REGION Network 2: 0 - Запуск системы с нуля
   RUNG wire#powerrail
      Contact( #Start )
      { S7_Templates := "SrcType := Int" } EQ_Contact(in1 := #"Step", in2 := 0)
      wire#w1
      S_Coil( "PS_StartUp_DB".Start )
      wire#w2
      Contact( "PS_StartUp_DB".Ready )
      Add(in1 := #"Step", in2 := 1, out => #"Step")
      { S7_Templates := "SrcType := Int" } EQ_Contact(in1 := #Mode, in2 := 0)
      S_Coil( "PID_PE_DB".Start )
   END_RUNG
   RUNG wire#w2
      { S7_Templates := "SrcType := Int" } GT_Contact(in1 := "PS_StartUp_DB"."Step", in2 := 0)
      wire#w3
      { S7_Templates := "SrcType := Int" } EQ_Contact(in1 := #Mode, in2 := 1)
      S_Coil( "PID_LE_in_DB".Start )
   END_RUNG
   RUNG wire#w3
      { S7_Templates := "SrcType := Int" } EQ_Contact(in1 := #Mode, in2 := 2)
      S_Coil( "PID_LE_out_DB".Start )
   END_RUNG
   RUNG wire#w1
      { S7_Templates := "SrcType := Int" } EQ_Contact(in1 := #Mode, in2 := 0)
      Move(in := #PE_StartUp, out1 => #PE_Work)
      wire#w4
      { S7_Templates := "SrcType := Int" } GE_Contact(in1 := "PS_StartUp_DB"."Step", in2 := 1)
      R_Coil( "PID_PE_DB".CMD.Force )
   END_RUNG
   RUNG wire#w4
      { S7_Templates := "SrcType := Int" } LT_Contact(in1 := "PS_StartUp_DB"."Step", in2 := 1)
      Move(in := "PS_Main_DB".PS_SP_Hz, out1 => "PID_PE_DB".PID_Hand)
      S_Coil( "PID_PE_DB".CMD.Force )
   END_RUNG
   RUNG wire#w1
      { S7_Templates := "SrcType := Int" } LT_Contact(in1 := #PS_cnt, in2 := #PS_REQ)
      Move(in := "PS_Main_DB".PS_CMD, out1 => #PS_cnt, out2 => #PS_REQ)
   END_RUNG
   // the same network as SCL:
   #_w1 := #Start AND (#"Step" = 0);
   IF #_w1 THEN "PS_StartUp_DB".Start := TRUE; END_IF;
   #_w2 := #_w1 AND "PS_StartUp_DB".Ready;
   IF #_w2 THEN #"Step" := #"Step" + 1; END_IF;
   IF #_w2 AND (#Mode = 0) THEN "PID_PE_DB".Start := TRUE; END_IF;
   #_w3 := #_w1 AND ("PS_StartUp_DB"."Step" > 0);
   IF #_w3 AND (#Mode = 1) THEN "PID_LE_in_DB".Start := TRUE; END_IF;
   IF #_w3 AND (#Mode = 2) THEN "PID_LE_out_DB".Start := TRUE; END_IF;
   #_w4 := #_w1 AND (#Mode = 0);
   IF #_w4 THEN #PE_Work := #PE_StartUp; END_IF;
   IF #_w4 AND ("PS_StartUp_DB"."Step" >= 1) THEN "PID_PE_DB".CMD.Force := FALSE; END_IF;
   IF #_w4 AND ("PS_StartUp_DB"."Step" < 1) THEN
       "PID_PE_DB".PID_Hand := "PS_Main_DB".PS_SP_Hz;
       "PID_PE_DB".CMD.Force := TRUE;
   END_IF;
   IF #_w1 AND (#PS_cnt < #PS_REQ) THEN
       #PS_cnt := "PS_Main_DB".PS_CMD;
       #PS_REQ := "PS_Main_DB".PS_CMD;
   END_IF;
END_REGION

REGION Network 3: 1 - Штатная работа системы
   RUNG wire#powerrail
      { S7_Templates := "SrcType := Int" } EQ_Contact(in1 := #"Step", in2 := 1)
      { S7_Templates := "SrcType := Int" } LE_Contact(in1 := #Mode, in2 := 2)
      wire#w1
      { S7_Templates := "SrcType := Real" } GE_Contact(in1 := #SP_Hz, in2 := #SP_High)
      { S7_Templates := "SrcType := Int" } EQ_Contact(in1 := #PS_REQ, in2 := #PS_cnt)
      wire#w2
      { S7_Templates := "SrcType := Int" } LT_Contact(in1 := "PS_Main_DB".PS_CMD, in2 := "PS_Main_DB".PS_Group)
      { S7_Templates := "SrcType := Int" } LT_Contact(in1 := #PS_REQ, in2 := "PS_Main_DB".PS_Group)
      { S7_Templates := "SrcType := Int" } EQ_Contact(in1 := "PS_cnt_DB"."Step", in2 := 10)
      Coil( #T_Delay_ADD.Start )
      Contact( #T_Delay_ADD."Exit" )
      Add(in1 := #PS_REQ, in2 := 1, out => #PS_REQ)
   END_RUNG
   RUNG wire#w2
      I_Contact( #Reload )
      I_Contact( #Load )
      I_Contact( #Rotation )
      I_Contact( #Deload )
      I_Contact( #T_Delay_ADD."Exit" )
      { S7_Templates := "SrcType := Int" } EQ_Contact(in1 := "PS_cnt_DB"."Step", in2 := 10)
      Coil( #T_Delay_SUB.Start )
      Contact( #T_Delay_SUB."Exit" )
      wire#w3
      { S7_Templates := "SrcType := Int" } GT_Contact(in1 := #PS_REQ, in2 := "PS_Main_DB".PS_CMD)
      S_Coil( #Reload )
   END_RUNG
   RUNG wire#w3
      { S7_Templates := "SrcType := Int" } GT_Contact(in1 := "PS_Main_DB".PS_CMD, in2 := #PS_REQ)
      S_Coil( #Deload )
   END_RUNG
   RUNG wire#w1
      { S7_Templates := "SrcType := Real" } LT_Contact(in1 := #SP_Hz, in2 := #SP_Low)
      { S7_Templates := "SrcType := Int" } EQ_Contact(in1 := #PS_REQ, in2 := #PS_cnt)
      { S7_Templates := "SrcType := Int" } GT_Contact(in1 := #PS_REQ, in2 := 1)
      { S7_Templates := "SrcType := Int" } EQ_Contact(in1 := "PS_cnt_DB"."Step", in2 := 10)
      Sub(in1 := #PS_REQ, in2 := 1, out => #PS_REQ)
   END_RUNG
   RUNG wire#w1
      Move(in := #PE_SP, out1 => #PE_Work)
   END_RUNG
   // the same network as SCL:
   #_w1 := (#"Step" = 1) AND (#Mode <= 2);
   #_w2 := #_w1 AND (#SP_Hz >= #SP_High) AND (#PS_REQ = #PS_cnt);
   #T_Delay_ADD.Start := #_w2 AND ("PS_Main_DB".PS_CMD < "PS_Main_DB".PS_Group) AND (#PS_REQ < "PS_Main_DB".PS_Group) AND ("PS_cnt_DB"."Step" = 10);
   IF #T_Delay_ADD.Start AND #T_Delay_ADD."Exit" THEN #PS_REQ := #PS_REQ + 1; END_IF;
   #T_Delay_SUB.Start := #_w2 AND NOT #Reload AND NOT #Load AND NOT #Rotation AND NOT #Deload AND NOT #T_Delay_ADD."Exit" AND ("PS_cnt_DB"."Step" = 10);
   #_w3 := #T_Delay_SUB.Start AND #T_Delay_SUB."Exit";
   IF #_w3 AND (#PS_REQ > "PS_Main_DB".PS_CMD) THEN #Reload := TRUE; END_IF;
   IF #_w3 AND ("PS_Main_DB".PS_CMD > #PS_REQ) THEN #Deload := TRUE; END_IF;
   IF #_w1 AND (#SP_Hz < #SP_Low) AND (#PS_REQ = #PS_cnt) AND (#PS_REQ > 1) AND ("PS_cnt_DB"."Step" = 10) THEN
       #PS_REQ := #PS_REQ - 1;
   END_IF;
   IF #_w1 THEN #PE_Work := #PE_SP; END_IF;
END_REGION

REGION Network 4: 1 - Штатная работа - макс производительность
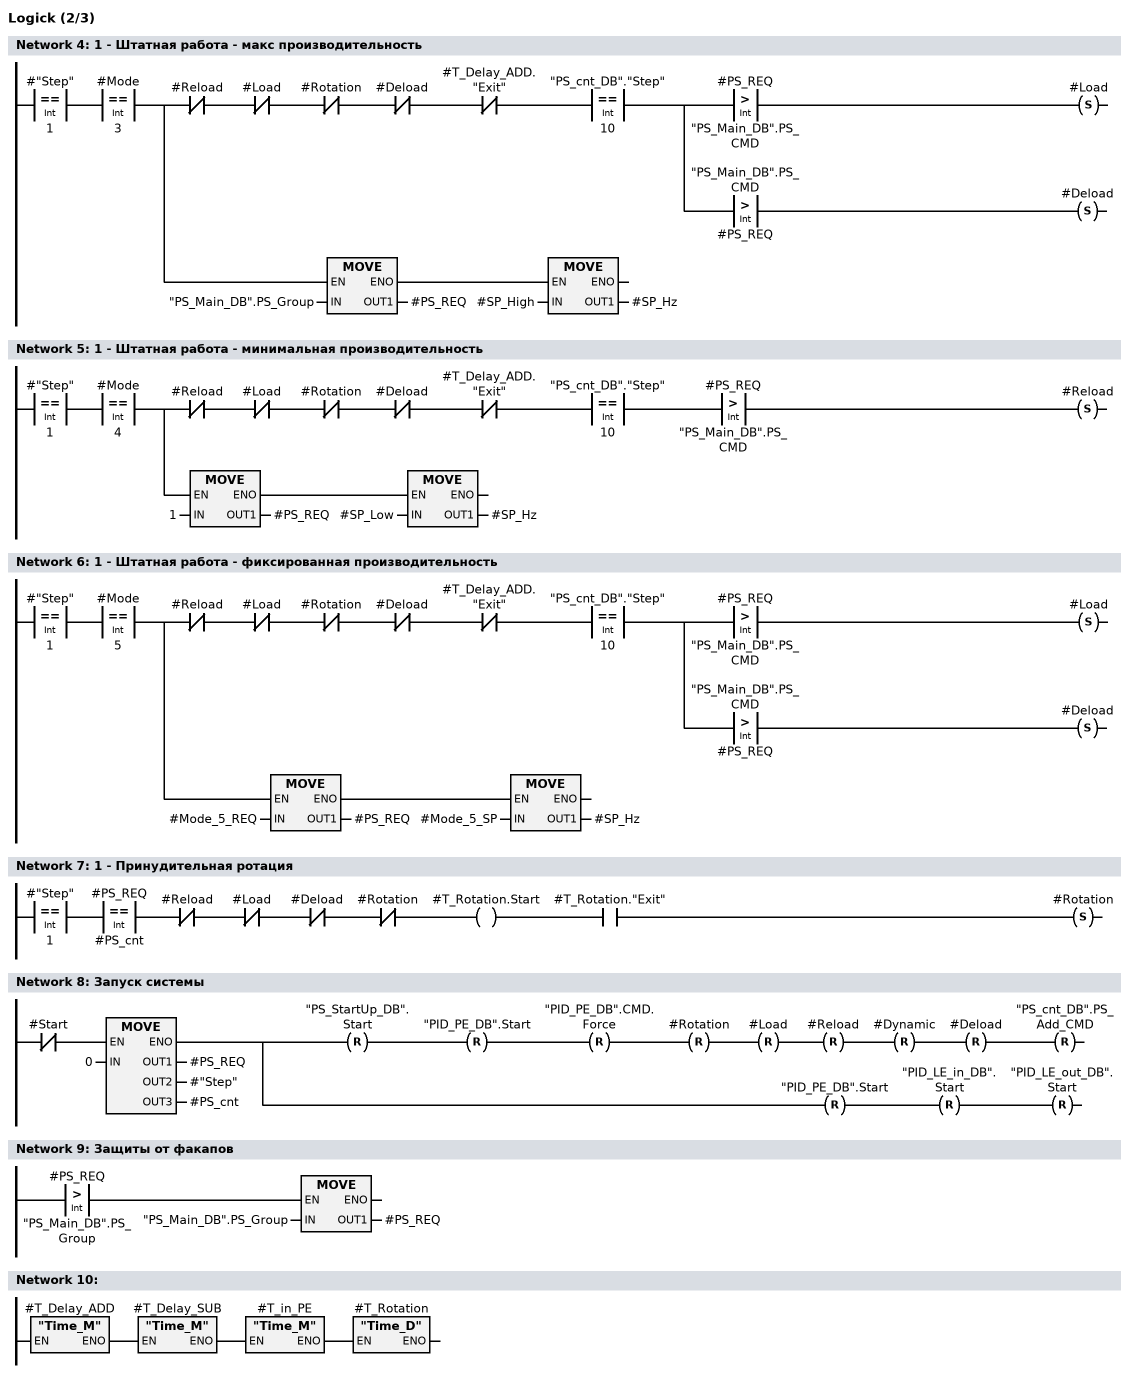
   RUNG wire#powerrail
      { S7_Templates := "SrcType := Int" } EQ_Contact(in1 := #"Step", in2 := 1)
      { S7_Templates := "SrcType := Int" } EQ_Contact(in1 := #Mode, in2 := 3)
      wire#w1
      I_Contact( #Reload )
      I_Contact( #Load )
      I_Contact( #Rotation )
      I_Contact( #Deload )
      I_Contact( #T_Delay_ADD."Exit" )
      { S7_Templates := "SrcType := Int" } EQ_Contact(in1 := "PS_cnt_DB"."Step", in2 := 10)
      wire#w2
      { S7_Templates := "SrcType := Int" } GT_Contact(in1 := #PS_REQ, in2 := "PS_Main_DB".PS_CMD)
      S_Coil( #Load )
   END_RUNG
   RUNG wire#w2
      { S7_Templates := "SrcType := Int" } GT_Contact(in1 := "PS_Main_DB".PS_CMD, in2 := #PS_REQ)
      S_Coil( #Deload )
   END_RUNG
   RUNG wire#w1
      Move(in := "PS_Main_DB".PS_Group, out1 => #PS_REQ)
      Move(in := #SP_High, out1 => #SP_Hz)
   END_RUNG
   // the same network as SCL:
   #_w1 := (#"Step" = 1) AND (#Mode = 3);
   #_w2 := #_w1 AND NOT #Reload AND NOT #Load AND NOT #Rotation AND NOT #Deload AND NOT #T_Delay_ADD."Exit" AND ("PS_cnt_DB"."Step" = 10);
   IF #_w2 AND (#PS_REQ > "PS_Main_DB".PS_CMD) THEN #Load := TRUE; END_IF;
   IF #_w2 AND ("PS_Main_DB".PS_CMD > #PS_REQ) THEN #Deload := TRUE; END_IF;
   IF #_w1 THEN
       #PS_REQ := "PS_Main_DB".PS_Group;
       #SP_Hz := #SP_High;
   END_IF;
END_REGION

REGION Network 5: 1 - Штатная работа - минимальная производительность
   RUNG wire#powerrail
      { S7_Templates := "SrcType := Int" } EQ_Contact(in1 := #"Step", in2 := 1)
      { S7_Templates := "SrcType := Int" } EQ_Contact(in1 := #Mode, in2 := 4)
      wire#w1
      I_Contact( #Reload )
      I_Contact( #Load )
      I_Contact( #Rotation )
      I_Contact( #Deload )
      I_Contact( #T_Delay_ADD."Exit" )
      { S7_Templates := "SrcType := Int" } EQ_Contact(in1 := "PS_cnt_DB"."Step", in2 := 10)
      { S7_Templates := "SrcType := Int" } GT_Contact(in1 := #PS_REQ, in2 := "PS_Main_DB".PS_CMD)
      S_Coil( #Reload )
   END_RUNG
   RUNG wire#w1
      Move(in := 1, out1 => #PS_REQ)
      Move(in := #SP_Low, out1 => #SP_Hz)
   END_RUNG
   // the same network as SCL:
   #_w1 := (#"Step" = 1) AND (#Mode = 4);
   IF #_w1 AND NOT #Reload AND NOT #Load AND NOT #Rotation AND NOT #Deload AND NOT #T_Delay_ADD."Exit" AND ("PS_cnt_DB"."Step" = 10) AND (#PS_REQ > "PS_Main_DB".PS_CMD) THEN
       #Reload := TRUE;
   END_IF;
   IF #_w1 THEN
       #PS_REQ := 1;
       #SP_Hz := #SP_Low;
   END_IF;
END_REGION

REGION Network 6: 1 - Штатная работа - фиксированная производительность
   RUNG wire#powerrail
      { S7_Templates := "SrcType := Int" } EQ_Contact(in1 := #"Step", in2 := 1)
      { S7_Templates := "SrcType := Int" } EQ_Contact(in1 := #Mode, in2 := 5)
      wire#w1
      I_Contact( #Reload )
      I_Contact( #Load )
      I_Contact( #Rotation )
      I_Contact( #Deload )
      I_Contact( #T_Delay_ADD."Exit" )
      { S7_Templates := "SrcType := Int" } EQ_Contact(in1 := "PS_cnt_DB"."Step", in2 := 10)
      wire#w2
      { S7_Templates := "SrcType := Int" } GT_Contact(in1 := #PS_REQ, in2 := "PS_Main_DB".PS_CMD)
      S_Coil( #Load )
   END_RUNG
   RUNG wire#w2
      { S7_Templates := "SrcType := Int" } GT_Contact(in1 := "PS_Main_DB".PS_CMD, in2 := #PS_REQ)
      S_Coil( #Deload )
   END_RUNG
   RUNG wire#w1
      Move(in := #Mode_5_REQ, out1 => #PS_REQ)
      Move(in := #Mode_5_SP, out1 => #SP_Hz)
   END_RUNG
   // the same network as SCL:
   #_w1 := (#"Step" = 1) AND (#Mode = 5);
   #_w2 := #_w1 AND NOT #Reload AND NOT #Load AND NOT #Rotation AND NOT #Deload AND NOT #T_Delay_ADD."Exit" AND ("PS_cnt_DB"."Step" = 10);
   IF #_w2 AND (#PS_REQ > "PS_Main_DB".PS_CMD) THEN #Load := TRUE; END_IF;
   IF #_w2 AND ("PS_Main_DB".PS_CMD > #PS_REQ) THEN #Deload := TRUE; END_IF;
   IF #_w1 THEN
       #PS_REQ := #Mode_5_REQ;
       #SP_Hz := #Mode_5_SP;
   END_IF;
END_REGION

REGION Network 7: 1 - Принудительная ротация
   RUNG wire#powerrail
      { S7_Templates := "SrcType := Int" } EQ_Contact(in1 := #"Step", in2 := 1)
      { S7_Templates := "SrcType := Int" } EQ_Contact(in1 := #PS_REQ, in2 := #PS_cnt)
      I_Contact( #Reload )
      I_Contact( #Load )
      I_Contact( #Deload )
      I_Contact( #Rotation )
      Coil( #T_Rotation.Start )
      Contact( #T_Rotation."Exit" )
      S_Coil( #Rotation )
   END_RUNG
   // the same network as SCL:
   #T_Rotation.Start := (#"Step" = 1) AND (#PS_REQ = #PS_cnt) AND NOT #Reload AND NOT #Load AND NOT #Deload AND NOT #Rotation;
   IF #T_Rotation.Start AND #T_Rotation."Exit" THEN #Rotation := TRUE; END_IF;
END_REGION

REGION Network 8: Запуск системы
   RUNG wire#powerrail
      I_Contact( #Start )
      Move(in := 0, out1 => #PS_REQ, out2 => #"Step", out3 => #PS_cnt)
      wire#w1
      R_Coil( "PS_StartUp_DB".Start )
      R_Coil( "PID_PE_DB".Start )
      R_Coil( "PID_PE_DB".CMD.Force )
      R_Coil( #Rotation )
      R_Coil( #Load )
      R_Coil( #Reload )
      R_Coil( #Dynamic )
      R_Coil( #Deload )
      R_Coil( "PS_cnt_DB".PS_Add_CMD )
   END_RUNG
   RUNG wire#w1
      R_Coil( "PID_PE_DB".Start )
      R_Coil( "PID_LE_in_DB".Start )
      R_Coil( "PID_LE_out_DB".Start )
   END_RUNG
   // the same network as SCL:
   IF NOT #Start THEN
       #PS_REQ := 0;
       #"Step" := 0;
       #PS_cnt := 0;
       "PS_StartUp_DB".Start := FALSE;
       "PID_PE_DB".Start := FALSE;
       "PID_PE_DB".CMD.Force := FALSE;
       #Rotation := FALSE;
       #Load := FALSE;
       #Reload := FALSE;
       #Dynamic := FALSE;
       #Deload := FALSE;
       "PS_cnt_DB".PS_Add_CMD := FALSE;
       "PID_PE_DB".Start := FALSE;
       "PID_LE_in_DB".Start := FALSE;
       "PID_LE_out_DB".Start := FALSE;
   END_IF;
END_REGION

REGION Network 9: Защиты от факапов
   RUNG wire#powerrail
      { S7_Templates := "SrcType := Int" } GT_Contact(in1 := #PS_REQ, in2 := "PS_Main_DB".PS_Group)
      Move(in := "PS_Main_DB".PS_Group, out1 => #PS_REQ)
   END_RUNG
   // the same network as SCL:
   IF #PS_REQ > "PS_Main_DB".PS_Group THEN #PS_REQ := "PS_Main_DB".PS_Group; END_IF;
END_REGION

REGION Network 10
   RUNG wire#powerrail
      #T_Delay_ADD()
      #T_Delay_SUB()
      #T_in_PE()
      #T_Rotation()
   END_RUNG
   // the same network as SCL:
   #T_Delay_ADD(ENO => #_w1);   // "Time_M"
   #T_Delay_SUB(EN := #_w1, ENO => #_w2);   // "Time_M"
   #T_in_PE(EN := #_w2, ENO => #_w3);   // "Time_M"
   IF #_w3 THEN
       #T_Rotation();   // "Time_D"
   END_IF;
END_REGION

REGION Network 11: Соотношение давления к уставке
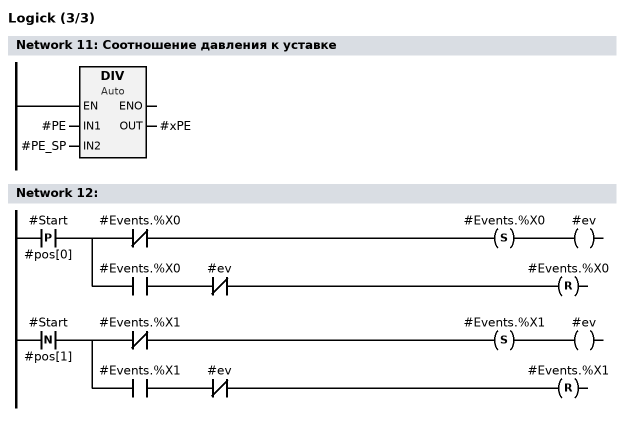
   RUNG wire#powerrail
      Div(in1 := #PE, in2 := #PE_SP, out => #xPE)
   END_RUNG
   // the same network as SCL:
   #xPE := #PE / #PE_SP;
END_REGION

REGION Network 12
   RUNG wire#powerrail
      P_Contact(operand := #Start, bit := #pos[0])
      wire#w1
      I_Contact( #Events.%X0 )
      S_Coil( #Events.%X0 )
      Coil( #ev )
   END_RUNG
   RUNG wire#w1
      Contact( #Events.%X0 )
      I_Contact( #ev )
      R_Coil( #Events.%X0 )
   END_RUNG
   RUNG wire#powerrail
      N_Contact(operand := #Start, bit := #pos[1])
      wire#w2
      I_Contact( #Events.%X1 )
      S_Coil( #Events.%X1 )
      Coil( #ev )
   END_RUNG
   RUNG wire#w2
      Contact( #Events.%X1 )
      I_Contact( #ev )
      R_Coil( #Events.%X1 )
   END_RUNG
   // the same network as SCL:
   #_w1 := #Start AND NOT #pos[0];   // rising edge of #Start
   #pos[0] := #Start;
   #_w2 := #_w1 AND NOT #Events.%X0;
   IF #_w2 THEN #Events.%X0 := TRUE; END_IF;
   #ev := #_w2;
   IF #_w1 AND #Events.%X0 AND NOT #ev THEN #Events.%X0 := FALSE; END_IF;
   #_w3 := NOT #Start AND #pos[1];   // falling edge of #Start
   #pos[1] := #Start;
   #_w4 := #_w3 AND NOT #Events.%X1;
   IF #_w4 THEN #Events.%X1 := TRUE; END_IF;
   #ev := #_w4;
   IF #_w3 AND #Events.%X1 AND NOT #ev THEN #Events.%X1 := FALSE; END_IF;
END_REGION
END_FUNCTION_BLOCK

FUNCTION_BLOCK "PS_Main"   // FB10, LAD
{ S7_Optimized_Access := 'FALSE' }
VERSION : 0.1
// stored: AutoNumber false, IsIECCheckEnabled false, SetENOAutomatically false, UDAEnableTagReadback false
   VAR_IN_OUT
      PS_REQ : Int;   // Требуемуе кол-во насосов
      PS_cnt : Int;
   END_VAR
   VAR DB_SPECIFIC
      Step_Up { S7_SetPoint := 'True'} : Array[1..6] of Real;   // Ускорения насоса, Гц/сек
      Step_Down { S7_SetPoint := 'True'} : Array[1..6] of Real;   // Замедление насоса, Гц/сек
   END_VAR
   VAR
      PS_One { S7_SetPoint := 'True'} : Array[0..10] of "PS_One";   // Pump System - One Pump
   END_VAR
   VAR DB_SPECIFIC
      PS_All { S7_SetPoint := 'True'} : Int := 7;   // Общее количество насосов
      PS_Group { S7_SetPoint := 'True'} : Int := 5;   // Число основных насосов
      PS_Reserv { S7_SetPoint := 'True'} : Int := 2;   // Число резервных насосов
      PS_Ready : Int;   // Число готовых насосов
      PS_CMD : Int;   // Число насосов в работе
      PS_Work : Int;   // Число штатно работающих насосов
      PS_Load : Int;   // Число нагруженных насосов
      PS_SP_Hz : Real;   // Уставка - штатная работа
      PS_Point : Real;
      PS_min_cnt : Int;   // Число замедленных насосов
   END_VAR
   VAR_TEMP   // added for the SCL form of the ladder/FBD networks
      _w1 : Bool;
   END_VAR
BEGIN

REGION Network 1: Распределение нагрузки по насосам
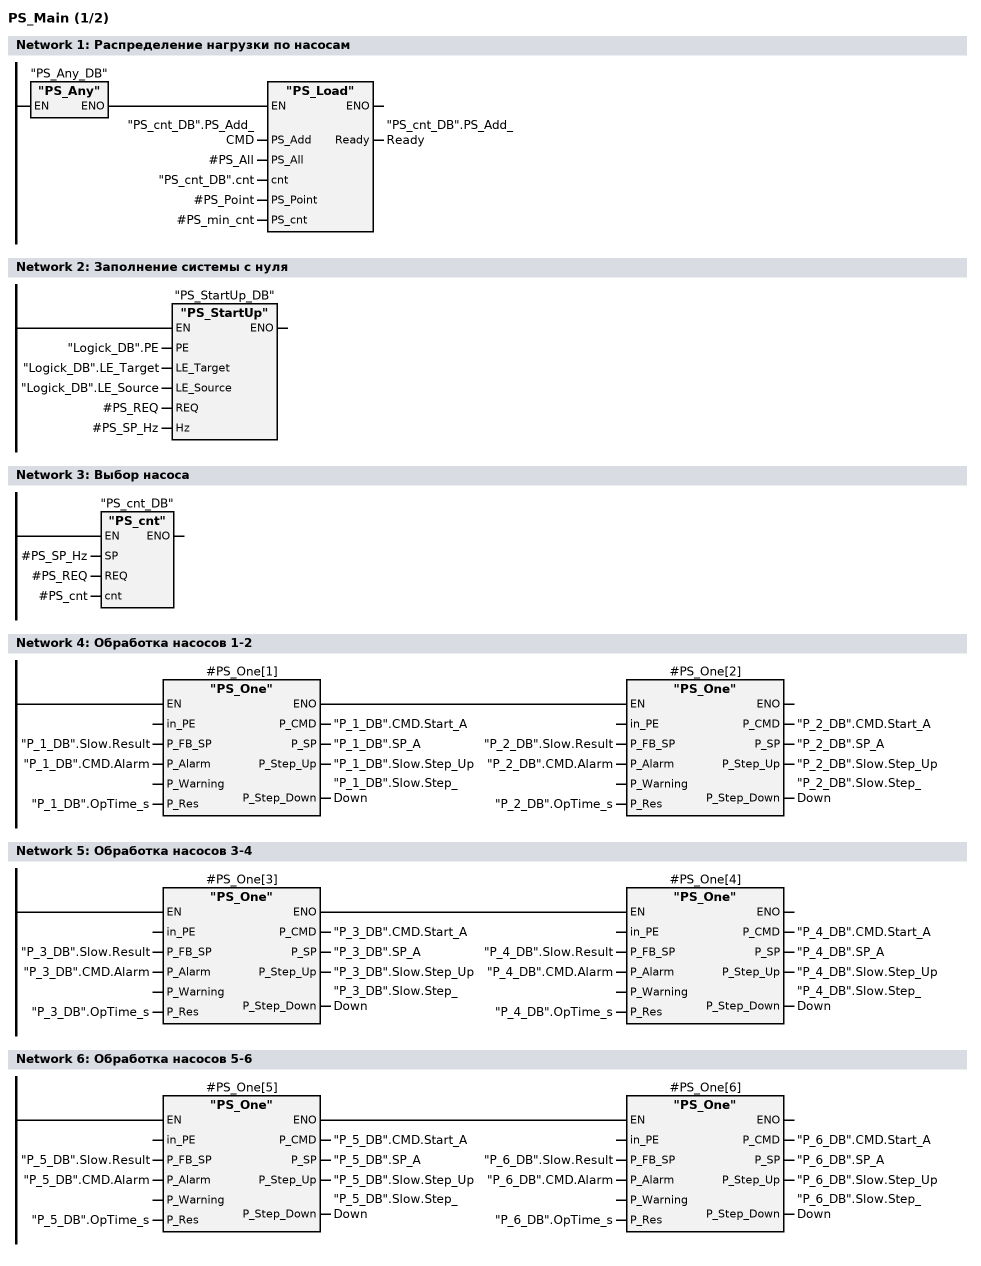
   RUNG wire#powerrail
      "PS_Any_DB"()
      "PS_Load"(PS_Add := "PS_cnt_DB".PS_Add_CMD, PS_All := #PS_All, cnt := "PS_cnt_DB".cnt, PS_Point := #PS_Point, PS_cnt := #PS_min_cnt, Ready => "PS_cnt_DB".PS_Add_Ready)
   END_RUNG
   // the same network as SCL:
   "PS_Any_DB"(ENO => #_w1);   // "PS_Any"
   IF #_w1 THEN
       "PS_Load"(PS_Add := "PS_cnt_DB".PS_Add_CMD,
                 PS_All := #PS_All,
                 cnt := "PS_cnt_DB".cnt,
                 PS_Point := #PS_Point,
                 PS_cnt := #PS_min_cnt,
                 Ready => "PS_cnt_DB".PS_Add_Ready);
   END_IF;
END_REGION

REGION Network 2: Заполнение системы с нуля
   RUNG wire#powerrail
      "PS_StartUp_DB"(PE := "Logick_DB".PE, LE_Target := "Logick_DB".LE_Target, LE_Source := "Logick_DB".LE_Source, REQ := #PS_REQ, Hz := #PS_SP_Hz)
   END_RUNG
   // the same network as SCL:
   "PS_StartUp_DB"(PE := "Logick_DB".PE,   // "PS_StartUp"
                   LE_Target := "Logick_DB".LE_Target,
                   LE_Source := "Logick_DB".LE_Source,
                   REQ := #PS_REQ,
                   Hz := #PS_SP_Hz);
END_REGION

REGION Network 3: Выбор насоса
   RUNG wire#powerrail
      "PS_cnt_DB"(SP := #PS_SP_Hz, REQ := #PS_REQ, cnt := #PS_cnt)
   END_RUNG
   // the same network as SCL:
   "PS_cnt_DB"(SP := #PS_SP_Hz, REQ := #PS_REQ, cnt := #PS_cnt);   // "PS_cnt"
END_REGION

REGION Network 4: Обработка насосов 1-2
   RUNG wire#powerrail
      #PS_One[1](in_PE :=, P_FB_SP := "P_1_DB".Slow.Result, P_Alarm := "P_1_DB".CMD.Alarm, P_Warning :=, P_Res := "P_1_DB".OpTime_s, P_CMD => "P_1_DB".CMD.Start_A, P_SP => "P_1_DB".SP_A, P_Step_Up => "P_1_DB".Slow.Step_Up, P_Step_Down => "P_1_DB".Slow.Step_Down)
      #PS_One[2](in_PE :=, P_FB_SP := "P_2_DB".Slow.Result, P_Alarm := "P_2_DB".CMD.Alarm, P_Warning :=, P_Res := "P_2_DB".OpTime_s, P_CMD => "P_2_DB".CMD.Start_A, P_SP => "P_2_DB".SP_A, P_Step_Up => "P_2_DB".Slow.Step_Up, P_Step_Down => "P_2_DB".Slow.Step_Down)
   END_RUNG
   // the same network as SCL:
   #PS_One[1](P_FB_SP := "P_1_DB".Slow.Result,   // "PS_One"
              P_Alarm := "P_1_DB".CMD.Alarm,
              P_Res := "P_1_DB".OpTime_s,
              P_CMD => "P_1_DB".CMD.Start_A,
              P_SP => "P_1_DB".SP_A,
              P_Step_Up => "P_1_DB".Slow.Step_Up,
              P_Step_Down => "P_1_DB".Slow.Step_Down,
              ENO => #_w1);
   IF #_w1 THEN
       #PS_One[2](P_FB_SP := "P_2_DB".Slow.Result,   // "PS_One"
                  P_Alarm := "P_2_DB".CMD.Alarm,
                  P_Res := "P_2_DB".OpTime_s,
                  P_CMD => "P_2_DB".CMD.Start_A,
                  P_SP => "P_2_DB".SP_A,
                  P_Step_Up => "P_2_DB".Slow.Step_Up,
                  P_Step_Down => "P_2_DB".Slow.Step_Down);
   END_IF;
END_REGION

REGION Network 5: Обработка насосов 3-4
   RUNG wire#powerrail
      #PS_One[3](in_PE :=, P_FB_SP := "P_3_DB".Slow.Result, P_Alarm := "P_3_DB".CMD.Alarm, P_Warning :=, P_Res := "P_3_DB".OpTime_s, P_CMD => "P_3_DB".CMD.Start_A, P_SP => "P_3_DB".SP_A, P_Step_Up => "P_3_DB".Slow.Step_Up, P_Step_Down => "P_3_DB".Slow.Step_Down)
      #PS_One[4](in_PE :=, P_FB_SP := "P_4_DB".Slow.Result, P_Alarm := "P_4_DB".CMD.Alarm, P_Warning :=, P_Res := "P_4_DB".OpTime_s, P_CMD => "P_4_DB".CMD.Start_A, P_SP => "P_4_DB".SP_A, P_Step_Up => "P_4_DB".Slow.Step_Up, P_Step_Down => "P_4_DB".Slow.Step_Down)
   END_RUNG
   // the same network as SCL:
   #PS_One[3](P_FB_SP := "P_3_DB".Slow.Result,   // "PS_One"
              P_Alarm := "P_3_DB".CMD.Alarm,
              P_Res := "P_3_DB".OpTime_s,
              P_CMD => "P_3_DB".CMD.Start_A,
              P_SP => "P_3_DB".SP_A,
              P_Step_Up => "P_3_DB".Slow.Step_Up,
              P_Step_Down => "P_3_DB".Slow.Step_Down,
              ENO => #_w1);
   IF #_w1 THEN
       #PS_One[4](P_FB_SP := "P_4_DB".Slow.Result,   // "PS_One"
                  P_Alarm := "P_4_DB".CMD.Alarm,
                  P_Res := "P_4_DB".OpTime_s,
                  P_CMD => "P_4_DB".CMD.Start_A,
                  P_SP => "P_4_DB".SP_A,
                  P_Step_Up => "P_4_DB".Slow.Step_Up,
                  P_Step_Down => "P_4_DB".Slow.Step_Down);
   END_IF;
END_REGION

REGION Network 6: Обработка насосов 5-6
   RUNG wire#powerrail
      #PS_One[5](in_PE :=, P_FB_SP := "P_5_DB".Slow.Result, P_Alarm := "P_5_DB".CMD.Alarm, P_Warning :=, P_Res := "P_5_DB".OpTime_s, P_CMD => "P_5_DB".CMD.Start_A, P_SP => "P_5_DB".SP_A, P_Step_Up => "P_5_DB".Slow.Step_Up, P_Step_Down => "P_5_DB".Slow.Step_Down)
      #PS_One[6](in_PE :=, P_FB_SP := "P_6_DB".Slow.Result, P_Alarm := "P_6_DB".CMD.Alarm, P_Warning :=, P_Res := "P_6_DB".OpTime_s, P_CMD => "P_6_DB".CMD.Start_A, P_SP => "P_6_DB".SP_A, P_Step_Up => "P_6_DB".Slow.Step_Up, P_Step_Down => "P_6_DB".Slow.Step_Down)
   END_RUNG
   // the same network as SCL:
   #PS_One[5](P_FB_SP := "P_5_DB".Slow.Result,   // "PS_One"
              P_Alarm := "P_5_DB".CMD.Alarm,
              P_Res := "P_5_DB".OpTime_s,
              P_CMD => "P_5_DB".CMD.Start_A,
              P_SP => "P_5_DB".SP_A,
              P_Step_Up => "P_5_DB".Slow.Step_Up,
              P_Step_Down => "P_5_DB".Slow.Step_Down,
              ENO => #_w1);
   IF #_w1 THEN
       #PS_One[6](P_FB_SP := "P_6_DB".Slow.Result,   // "PS_One"
                  P_Alarm := "P_6_DB".CMD.Alarm,
                  P_Res := "P_6_DB".OpTime_s,
                  P_CMD => "P_6_DB".CMD.Start_A,
                  P_SP => "P_6_DB".SP_A,
                  P_Step_Up => "P_6_DB".Slow.Step_Up,
                  P_Step_Down => "P_6_DB".Slow.Step_Down);
   END_IF;
END_REGION

REGION Network 7: Обработка насосов 7-8
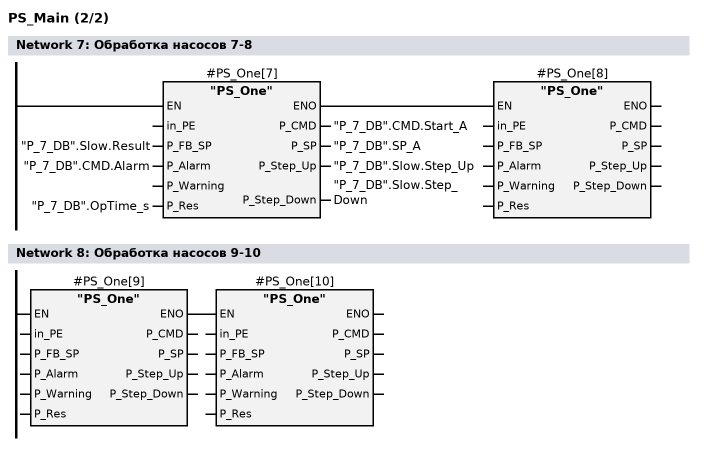
   RUNG wire#powerrail
      #PS_One[7](in_PE :=, P_FB_SP := "P_7_DB".Slow.Result, P_Alarm := "P_7_DB".CMD.Alarm, P_Warning :=, P_Res := "P_7_DB".OpTime_s, P_CMD => "P_7_DB".CMD.Start_A, P_SP => "P_7_DB".SP_A, P_Step_Up => "P_7_DB".Slow.Step_Up, P_Step_Down => "P_7_DB".Slow.Step_Down)
      #PS_One[8](in_PE :=, P_FB_SP :=, P_Alarm :=, P_Warning :=, P_Res :=, P_CMD =>, P_SP =>, P_Step_Up =>, P_Step_Down =>)
   END_RUNG
   // the same network as SCL:
   #PS_One[7](P_FB_SP := "P_7_DB".Slow.Result,   // "PS_One"
              P_Alarm := "P_7_DB".CMD.Alarm,
              P_Res := "P_7_DB".OpTime_s,
              P_CMD => "P_7_DB".CMD.Start_A,
              P_SP => "P_7_DB".SP_A,
              P_Step_Up => "P_7_DB".Slow.Step_Up,
              P_Step_Down => "P_7_DB".Slow.Step_Down,
              ENO => #_w1);
   IF #_w1 THEN
       #PS_One[8]();   // "PS_One"
   END_IF;
END_REGION

REGION Network 8: Обработка насосов 9-10
   RUNG wire#powerrail
      #PS_One[9](P_FB_SP :=, P_Alarm :=, P_Warning :=, P_Res :=, P_CMD =>, P_SP =>, P_Step_Up =>, P_Step_Down =>, in_PE :=)
      #PS_One[10](P_FB_SP :=, P_Alarm :=, P_Warning :=, P_Res :=, P_CMD =>, P_SP =>, P_Step_Up =>, P_Step_Down =>, in_PE :=)
   END_RUNG
   // the same network as SCL:
   #PS_One[9](ENO => #_w1);   // "PS_One"
   IF #_w1 THEN
       #PS_One[10]();   // "PS_One"
   END_IF;
END_REGION
END_FUNCTION_BLOCK

FUNCTION_BLOCK "PS_Any"
{ S7_Optimized_Access := 'FALSE' }
VERSION : 0.1
   VAR 
      x : Array[0..10] of Real;
      Delta_PE : Real;
      Delta_LE_in : Real;
      Delta_LE_out : Real;
   END_VAR


BEGIN
	//чтение уставки с ПИД-регулятора, если он в работе - режим работы по давлению
	IF "PID_PE_DB".Start AND NOT "PID_PE_DB".CMD.Hand AND "Logick_DB".Mode = 0 THEN
	    "Logick_DB".SP_Hz := "PID_PE_DB".Result;
	END_IF;
	
	//чтение уставки с ПИД-регулятора, если он в работе - режим работы по уровню в РЧВ
	IF "PID_LE_in_DB".Start AND NOT "PID_LE_in_DB".CMD.Hand AND "Logick_DB".Mode = 1 THEN
	    "Logick_DB".SP_Hz := "PID_LE_in_DB".Result;
	    IF "PS_StartUp_DB".Step = 1 THEN
	        "Logick_DB".SP_Hz := "Logick_DB".SP_Hz * "PS_StartUp_DB".xTime[2].Progress;
	    END_IF;
	END_IF;
	
	//чтение уставки с ПИД-регулятора, если он в работе - режим работы по уровню в городе
	IF "PID_LE_out_DB".Start AND NOT "PID_LE_out_DB".CMD.Hand AND "Logick_DB".Mode = 2 THEN
	    "Logick_DB".SP_Hz := "PID_LE_out_DB".Result;
	    IF "PS_StartUp_DB".Step = 1 THEN
	        "Logick_DB".SP_Hz := "Logick_DB".SP_Hz * "PS_StartUp_DB".xTime[2].Progress;
	    END_IF;
	END_IF;
	
	//рассчёт коррекции при превышении рабочего давления
	#x[1] := "Logick_DB".SP_PE_Alarm - "Logick_DB".SP_PE_Warning;
	#x[2] := "Logick_DB".PE - "Logick_DB".SP_PE_Warning;
	#x[3] := #x[2] / #x[1];
	#Delta_PE := 1 - #x[3];
	
	//давление выше рабочей точки
	IF #Delta_PE <= 1.0 THEN
	    "Logick_DB".PE_Warning := TRUE;
	    "Logick_DB".Alarms.%X0 := TRUE;
	ELSE
	    "Logick_DB".PE_Warning := FALSE;
	    "Logick_DB".Alarms.%X0 := FALSE;
	    #Delta_PE := 1.0;
	END_IF;
	
	//давление в аварийной зоне
	IF #Delta_PE <= 0.0 THEN
	    "Logick_DB".PE_Alarm := TRUE;
	    "Logick_DB".Alarms.%X1 := TRUE;
	    #Delta_PE := 0.0;
	ELSE
	    "Logick_DB".PE_Alarm := FALSE;
	END_IF;
	
	//рассчёт коррекции при падении уровня в РЧВ
	#x[4] := "Logick_DB".SP_LE_in_Warning - "Logick_DB".SP_LE_in_Alarm;
	#x[5] := "Logick_DB".LE_Source - "Logick_DB".SP_LE_in_Alarm;
	#x[6] := #x[5] / #x[4];
	#Delta_LE_in := #x[6];
	
	//уровень ниже рабочей точки
	IF #Delta_LE_in < 1.0 THEN
	    "Logick_DB".LE_in_Warning := TRUE;
	    "Logick_DB".Alarms.%X2 := TRUE;
	ELSE
	    "Logick_DB".LE_in_Warning := FALSE;
	    "Logick_DB".Alarms.%X2 := FALSE;
	    #Delta_LE_in := 1.0;
	END_IF;
	
	//уровень в аварийной зоне
	IF #Delta_LE_in <= 0.0 THEN
	    "Logick_DB".LE_in_Alarm := TRUE;
	    "Logick_DB".Alarms.%X3 := TRUE;
	    #Delta_LE_in := 0.0;
	ELSE
	    "Logick_DB".LE_in_Alarm := FALSE;
	END_IF;
	
	//рассчёт коррекции при превышении уровня в городе
	#x[7] := "Logick_DB".SP_LE_out_Alarm - "Logick_DB".SP_LE_out_Warning;
	#x[8] := "Logick_DB".LE_Target - "Logick_DB".SP_LE_out_Warning;
	#x[9] := #x[8] / #x[7];
	#Delta_LE_out := 1 - #x[9];
	
	//давление выше рабочей точки
	IF #Delta_LE_out <= 1.0 THEN
	    "Logick_DB".LE_out_Warning := TRUE;
	    "Logick_DB".Alarms.%X4 := TRUE;
	ELSE
	    "Logick_DB".LE_out_Warning := FALSE;
	    "Logick_DB".Alarms.%X4 := FALSE;
	    #Delta_LE_out := 1.0;
	END_IF;
	
	//давление в аварийной зоне
	IF #Delta_LE_out <= 0.0 THEN
	    "Logick_DB".LE_out_Alarm := TRUE;
	    "Logick_DB".Alarms.%X5 := TRUE;
	    #Delta_LE_out := 0.0;
	ELSE
	    "Logick_DB".LE_out_Alarm := FALSE;
	END_IF;
	
	//коррекция уставки при аварийных ситуациях
	"PS_Main_DB".PS_SP_Hz := "Logick_DB".SP_Hz * #Delta_PE * #Delta_LE_in * #Delta_LE_out;
	
	//Сброс аварий
	IF "Reset_All" THEN
	    "Logick_DB".Alarms := 0;
	END_IF;
	
	//индикатор аварий
	IF "Logick_DB".Alarms > 0 THEN
	    "Alm_Logick" := TRUE;
	END_IF;
	
END_FUNCTION_BLOCK

FUNCTION "PS_Load" : Void
{ S7_Optimized_Access := 'TRUE' }
VERSION : 0.1
   VAR_INPUT 
      PS_Add : Bool;
   END_VAR

   VAR_OUTPUT 
      Ready : Bool;
   END_VAR

   VAR_IN_OUT 
      PS_All : Int;
      cnt : Int;
      PS_Point : Real;   // точка схождения
      PS_cnt : Int;   // число готовых насосов
   END_VAR

   VAR_TEMP 
      x : Int;
   END_VAR


BEGIN
	//обнуление временных значений
	#PS_cnt := 0;
	#Ready := FALSE;
	"PS_cnt_DB".SP_High := "Logick_DB".SP_High;
	"PID_PE_DB".Settings.Max_out := "Logick_DB".SP_High + 1;
	"PID_PE_DB".Settings.Min_out := "Logick_DB".SP_Low - 1;
	"PID_LE_in_DB".Settings.Max_out := "Logick_DB".SP_High + 1;
	"PID_LE_in_DB".Settings.Min_out := "Logick_DB".SP_Low - 1;
	"PID_LE_out_DB".Settings.Max_out := "Logick_DB".SP_High + 1;
	"PID_LE_out_DB".Settings.Min_out := "Logick_DB".SP_Low - 1;
	"PS_cnt_DB".SP_Min := "Logick_DB".SP_Min;
	"Logick_DB".SP_Low := "PS_cnt_DB".SP_Low;
	"PS_Main_DB".PS_Ready := 0;
	"PS_Main_DB".PS_CMD := 0;
	"PS_Main_DB".PS_Work := 0;
	"PS_Main_DB".PS_Load := 0;
	
	IF "Logick_DB".SP_Hz > "Logick_DB".SP_High THEN
	    "Logick_DB".SP_Hz := "Logick_DB".SP_High;
	END_IF;
	
	//вычисление точки схождения скоростей
	#PS_Point := "PS_cnt_DB".SP_Low + ((("Logick_DB".SP_Hz - "PS_cnt_DB".SP_Low) / 3) * 2);
	
	//Распределение уставки по работающим насосам
	FOR #x := 1 TO #PS_All DO
	    
	    //число готовых насосов
	    IF "PS_Main_DB".PS_One[#x].CMD.Ready THEN
	        "PS_Main_DB".PS_Ready := "PS_Main_DB".PS_Ready + 1;
	    END_IF;
	    
	    //число насосов в работе
	    IF "PS_Main_DB".PS_One[#x].CMD.Start_M THEN
	        "PS_Main_DB".PS_CMD := "PS_Main_DB".PS_CMD + 1;
	    END_IF;
	    
	    //число насосов в штатном режиме
	    IF "PS_Main_DB".PS_One[#x].Status = 3 THEN
	        "PS_Main_DB".PS_Work := "PS_Main_DB".PS_Work + 1;
	    END_IF;
	    
	    //число насосов под нагрузкой
	    "PS_Main_DB".PS_Load := "PS_Main_DB".PS_Work + "PS_Main_DB".PS_min_cnt;
	    
	    
	    //запуск установки
	    IF "PS_cnt_DB".Step > 0 THEN
	        IF "PS_cnt_DB".Step < 10 OR "PS_cnt_DB".Step = 13 THEN
	            IF "PS_Main_DB".PS_One[#x].Status = 1 THEN
	                "PS_Main_DB".PS_One[#x].Mode := 2;
	            END_IF;
	            IF "PS_Main_DB".PS_One[#x].Status = 2 THEN
	                "PS_Main_DB".PS_One[#x].Mode := 3;
	            END_IF;
	            "PS_Main_DB".PS_One[#x].SP_A := "PS_cnt_DB".SP;
	        END_IF;
	    END_IF;
	    
	    //уставка в рабочем режиме
	    IF "PS_Main_DB".PS_One[#x].Status = 3 OR "PS_Main_DB".PS_One[#x].Status = 30 THEN
	        IF NOT "Logick_DB".PE_Warning AND NOT "Logick_DB".LE_in_Warning AND NOT "Logick_DB".LE_out_Warning THEN
	            "PS_Main_DB".PS_One[#x].SP_A := "Logick_DB".SP_Hz;
	        ELSE
	            "PS_Main_DB".PS_One[#x].SP_A := "PS_Main_DB".PS_SP_Hz;
	        END_IF;
	    END_IF;
	    
	  //цикл замедления при подключении нового насоса
	    IF #PS_Add THEN
	        
	        //команда замедлиться для подключения работающих насосов
	        IF "PS_Main_DB".PS_One[#x].Status = 3 THEN
	            "PS_Main_DB".PS_One[#x].Mode := 4;
	        END_IF;
	        
	        //коррекция уставки для замедленных насосов
	        IF "PS_Main_DB".PS_One[#x].Status = 40 THEN
	            "PS_Main_DB".PS_One[#x].SP_A := #PS_Point;
	        END_IF;
	        
	        //контроль готовности всех насосов
	        IF "PS_Main_DB".PS_One[#x].Status = 4 THEN
	            #PS_cnt := #PS_cnt + 1;
	            IF #PS_cnt = #cnt THEN
	                #Ready := true;
	            END_IF;
	        END_IF;
	        
	    END_IF;
	    
	    //возвращение в рабочий режим
	    IF NOT #PS_Add THEN
	        IF "PS_Main_DB".PS_One[#x].Status = 4 THEN
	            "PS_Main_DB".PS_One[#x].Mode := 3;
	        END_IF;
	    END_IF;
	    
	    //проброс уставок таймера по давлению
	    "PS_Main_DB".PS_One[#x].T_PE_Delay.SP_M := "Logick_DB".T_in_PE.SP_M;
	    "PS_Main_DB".PS_One[#x].T_PE_Delay.SP_S := "Logick_DB".T_in_PE.SP_S;
	    
	END_FOR;
	
END_FUNCTION

FUNCTION_BLOCK "PS_StartUp"   // FB13, LAD
{ S7_Optimized_Access := 'FALSE' }
VERSION : 0.1
// stored: AutoNumber false, IsIECCheckEnabled false, SetENOAutomatically false, UDAEnableTagReadback false
   VAR_INPUT
      PE : Real;
      LE_Target : Real;
      LE_Source : Real;
   END_VAR
   VAR_IN_OUT
      REQ : Int;
      Hz : Real;
   END_VAR
   VAR DB_SPECIFIC
      Start : Bool;   // Запуск системы
      Ready : Bool;   // Линия заполнена
      "Step" : Int;
      Warning : Word;
      PE_Point : Real;   // Давление на момент выхода плавный разгон
      PE_Delta : Real := 0.05;   // Допустимое отклонение
      PE_Min : Real;
      LE_Target_Point : Real;
      LE_Target_Delta : Real;
      LE_Target_Min : Real;
      LE_Source_Point : Real;
      LE_Source_Delta : Real;
      LE_Source_Min : Real;
      xSP : Array[0..5] of Struct
         Use { S7_SetPoint := 'True'} : Bool;
         REQ { S7_SetPoint := 'True'} : Int;
         Hz { S7_SetPoint := 'True'} : Real;
         PE { S7_SetPoint := 'True'} : Real;
         PE_Delta : Real;
      END_STRUCT;
   END_VAR
   VAR
      xTime { S7_SetPoint := 'True'} : Array[0..5] of "Time_M";
   END_VAR
   VAR_TEMP   // added for the SCL form of the ladder/FBD networks
      _w1 : Bool;
      _w2 : Bool;
      _w3 : Bool;
      _w4 : Bool;
      _w5 : Bool;
   END_VAR
BEGIN

REGION Network 1: 0 - Первичное заполнение труб
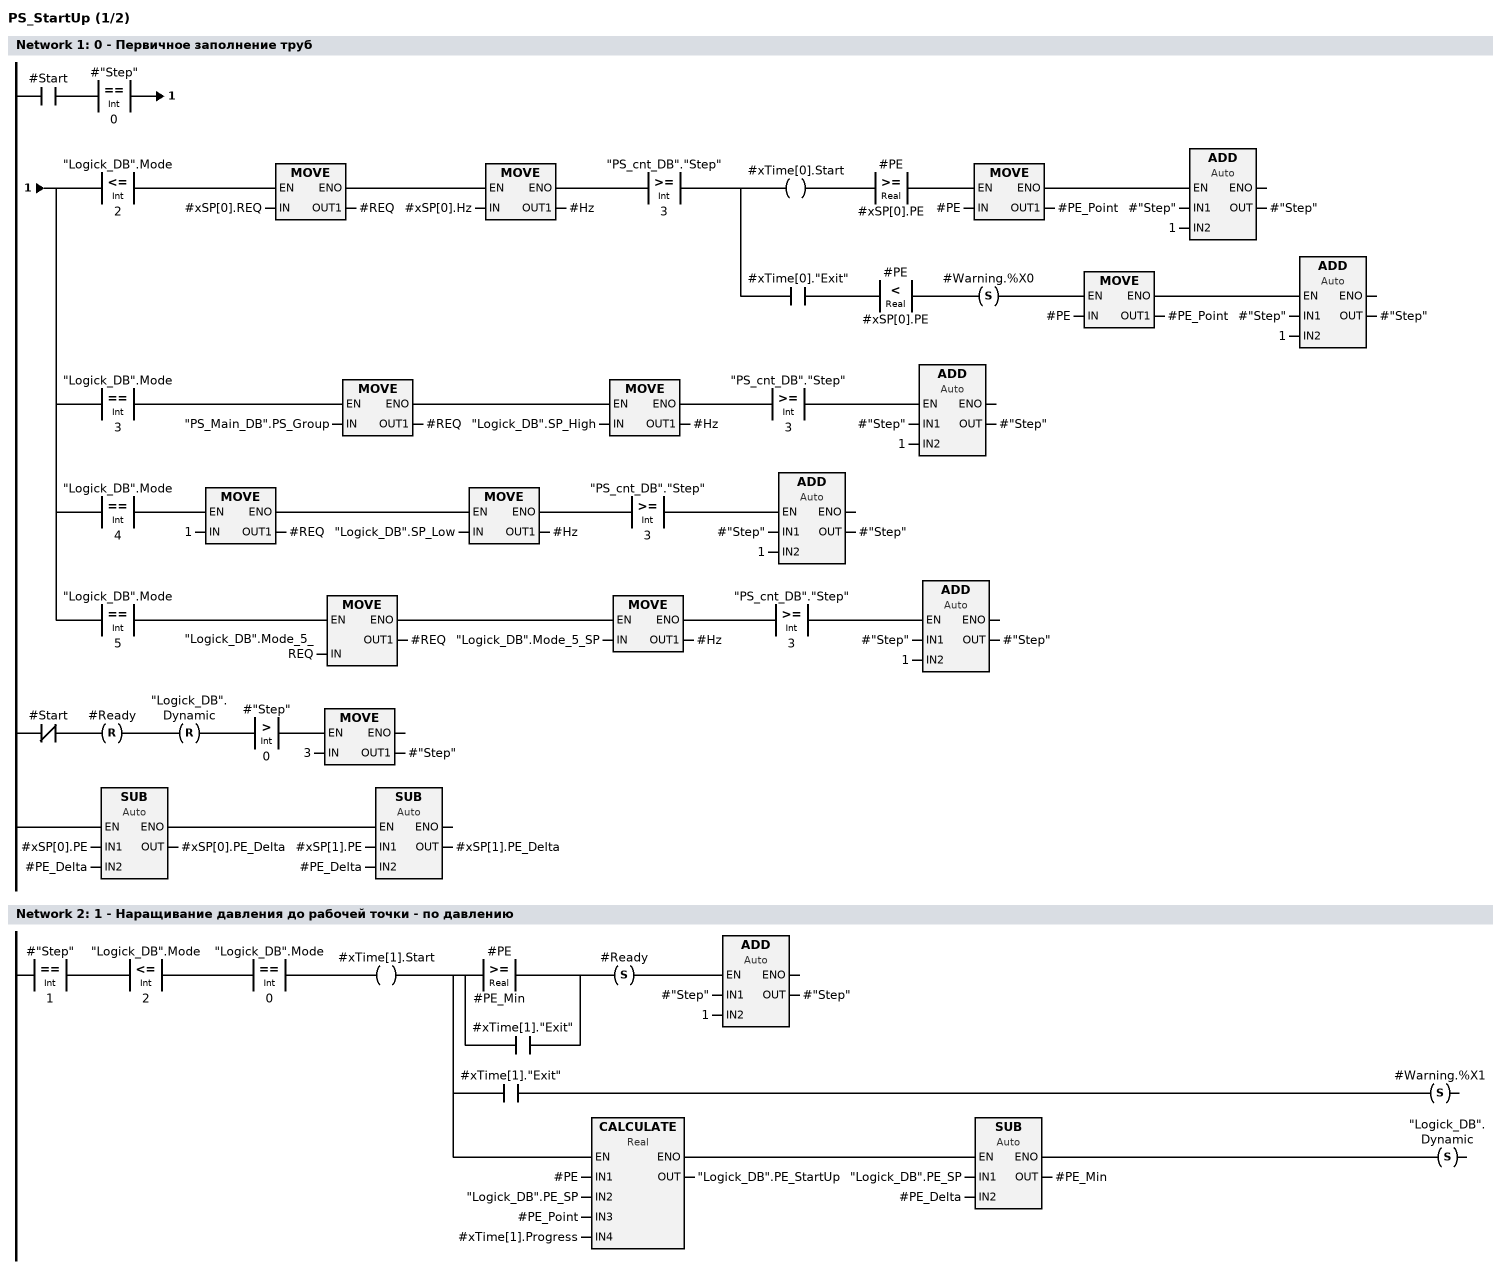
   RUNG wire#powerrail
      Contact( #Start )
      { S7_Templates := "SrcType := Int" } EQ_Contact(in1 := #"Step", in2 := 0)
      wire#w1
      { S7_Templates := "SrcType := Int" } LE_Contact(in1 := "Logick_DB".Mode, in2 := 2)
      Move(in := #xSP[0].REQ, out1 => #REQ)
      Move(in := #xSP[0].Hz, out1 => #Hz)
      { S7_Templates := "SrcType := Int" } GE_Contact(in1 := "PS_cnt_DB"."Step", in2 := 3)
      wire#w2
      Coil( #xTime[0].Start )
      { S7_Templates := "SrcType := Real" } GE_Contact(in1 := #PE, in2 := #xSP[0].PE)
      Move(in := #PE, out1 => #PE_Point)
      Add(in1 := #"Step", in2 := 1, out => #"Step")
   END_RUNG
   RUNG wire#w2
      Contact( #xTime[0]."Exit" )
      { S7_Templates := "SrcType := Real" } LT_Contact(in1 := #PE, in2 := #xSP[0].PE)
      S_Coil( #Warning.%X0 )
      Move(in := #PE, out1 => #PE_Point)
      Add(in1 := #"Step", in2 := 1, out => #"Step")
   END_RUNG
   RUNG wire#w1
      { S7_Templates := "SrcType := Int" } EQ_Contact(in1 := "Logick_DB".Mode, in2 := 3)
      Move(in := "PS_Main_DB".PS_Group, out1 => #REQ)
      Move(in := "Logick_DB".SP_High, out1 => #Hz)
      { S7_Templates := "SrcType := Int" } GE_Contact(in1 := "PS_cnt_DB"."Step", in2 := 3)
      Add(in1 := #"Step", in2 := 1, out => #"Step")
   END_RUNG
   RUNG wire#w1
      { S7_Templates := "SrcType := Int" } EQ_Contact(in1 := "Logick_DB".Mode, in2 := 4)
      Move(in := 1, out1 => #REQ)
      Move(in := "Logick_DB".SP_Low, out1 => #Hz)
      { S7_Templates := "SrcType := Int" } GE_Contact(in1 := "PS_cnt_DB"."Step", in2 := 3)
      Add(in1 := #"Step", in2 := 1, out => #"Step")
   END_RUNG
   RUNG wire#w1
      { S7_Templates := "SrcType := Int" } EQ_Contact(in1 := "Logick_DB".Mode, in2 := 5)
      Move(in := "Logick_DB".Mode_5_REQ, out1 => #REQ)
      Move(in := "Logick_DB".Mode_5_SP, out1 => #Hz)
      { S7_Templates := "SrcType := Int" } GE_Contact(in1 := "PS_cnt_DB"."Step", in2 := 3)
      Add(in1 := #"Step", in2 := 1, out => #"Step")
   END_RUNG
   RUNG wire#powerrail
      I_Contact( #Start )
      R_Coil( #Ready )
      R_Coil( "Logick_DB".Dynamic )
      { S7_Templates := "SrcType := Int" } GT_Contact(in1 := #"Step", in2 := 0)
      Move(in := 3, out1 => #"Step")
   END_RUNG
   RUNG wire#powerrail
      Sub(in1 := #xSP[0].PE, in2 := #PE_Delta, out => #xSP[0].PE_Delta)
      Sub(in1 := #xSP[1].PE, in2 := #PE_Delta, out => #xSP[1].PE_Delta)
   END_RUNG
   // the same network as SCL:
   #_w1 := #Start AND (#"Step" = 0);
   #_w2 := #_w1 AND ("Logick_DB".Mode <= 2);
   IF #_w2 THEN
       #REQ := #xSP[0].REQ;
       #Hz := #xSP[0].Hz;
   END_IF;
   #xTime[0].Start := #_w2 AND ("PS_cnt_DB"."Step" >= 3);
   IF #_w2 AND ("PS_cnt_DB"."Step" >= 3) AND (#PE >= #xSP[0].PE) THEN
       #PE_Point := #PE;
       #"Step" := #"Step" + 1;
   END_IF;
   IF #_w2 AND ("PS_cnt_DB"."Step" >= 3) AND #xTime[0]."Exit" AND (#PE < #xSP[0].PE) THEN
       #Warning.%X0 := TRUE;
       #PE_Point := #PE;
       #"Step" := #"Step" + 1;
   END_IF;
   #_w3 := #_w1 AND ("Logick_DB".Mode = 3);
   IF #_w3 THEN
       #REQ := "PS_Main_DB".PS_Group;
       #Hz := "Logick_DB".SP_High;
   END_IF;
   IF #_w3 AND ("PS_cnt_DB"."Step" >= 3) THEN #"Step" := #"Step" + 1; END_IF;
   #_w4 := #_w1 AND ("Logick_DB".Mode = 4);
   IF #_w4 THEN
       #REQ := 1;
       #Hz := "Logick_DB".SP_Low;
   END_IF;
   IF #_w4 AND ("PS_cnt_DB"."Step" >= 3) THEN #"Step" := #"Step" + 1; END_IF;
   #_w5 := #_w1 AND ("Logick_DB".Mode = 5);
   IF #_w5 THEN
       #REQ := "Logick_DB".Mode_5_REQ;
       #Hz := "Logick_DB".Mode_5_SP;
   END_IF;
   IF #_w5 AND ("PS_cnt_DB"."Step" >= 3) THEN #"Step" := #"Step" + 1; END_IF;
   IF NOT #Start THEN
       #Ready := FALSE;
       "Logick_DB".Dynamic := FALSE;
   END_IF;
   IF NOT #Start AND (#"Step" > 0) THEN #"Step" := 3; END_IF;
   #xSP[0].PE_Delta := #xSP[0].PE - #PE_Delta;
   #xSP[1].PE_Delta := #xSP[1].PE - #PE_Delta;
END_REGION

REGION Network 2: 1 - Наращивание давления до рабочей точки - по давлению
   RUNG wire#powerrail
      { S7_Templates := "SrcType := Int" } EQ_Contact(in1 := #"Step", in2 := 1)
      { S7_Templates := "SrcType := Int" } LE_Contact(in1 := "Logick_DB".Mode, in2 := 2)
      { S7_Templates := "SrcType := Int" } EQ_Contact(in1 := "Logick_DB".Mode, in2 := 0)
      Coil( #xTime[1].Start )
      wire#w1
      { S7_Templates := "SrcType := Real" } GE_Contact(in1 := #PE, in2 := #PE_Min)
      wire#w2
      S_Coil( #Ready )
      Add(in1 := #"Step", in2 := 1, out => #"Step")
   END_RUNG
   RUNG wire#w1
      Contact( #xTime[1]."Exit" )
   END_RUNG wire#w2
   RUNG wire#w1
      Contact( #xTime[1]."Exit" )
      S_Coil( #Warning.%X1 )
   END_RUNG
   RUNG wire#w1
      { S7_Templates := "SrcType := Real"; S7_Expression := "IN1 + (IN2 - IN3) * IN4" } Calculate(in1 := #PE, in2 := "Logick_DB".PE_SP, in3 := #PE_Point, in4 := #xTime[1].Progress, out => "Logick_DB".PE_StartUp)
      Sub(in1 := "Logick_DB".PE_SP, in2 := #PE_Delta, out => #PE_Min)
      S_Coil( "Logick_DB".Dynamic )
   END_RUNG
   // the same network as SCL:
   #xTime[1].Start := (#"Step" = 1) AND ("Logick_DB".Mode <= 2) AND ("Logick_DB".Mode = 0);
   #_w1 := (#"Step" = 1) AND ("Logick_DB".Mode <= 2) AND ("Logick_DB".Mode = 0);
   IF #_w1 AND ((#PE >= #PE_Min) OR #xTime[1]."Exit") THEN
       #Ready := TRUE;
       #"Step" := #"Step" + 1;
   END_IF;
   IF #_w1 AND #xTime[1]."Exit" THEN #Warning.%X1 := TRUE; END_IF;
   IF #_w1 THEN
       "Logick_DB".PE_StartUp := #PE + ("Logick_DB".PE_SP - #PE_Point) * #xTime[1].Progress;
       #PE_Min := "Logick_DB".PE_SP - #PE_Delta;
       "Logick_DB".Dynamic := TRUE;
   END_IF;
END_REGION

REGION Network 3: 1 - Наращивание давления до рабочей точки - по уровню в РЧВ
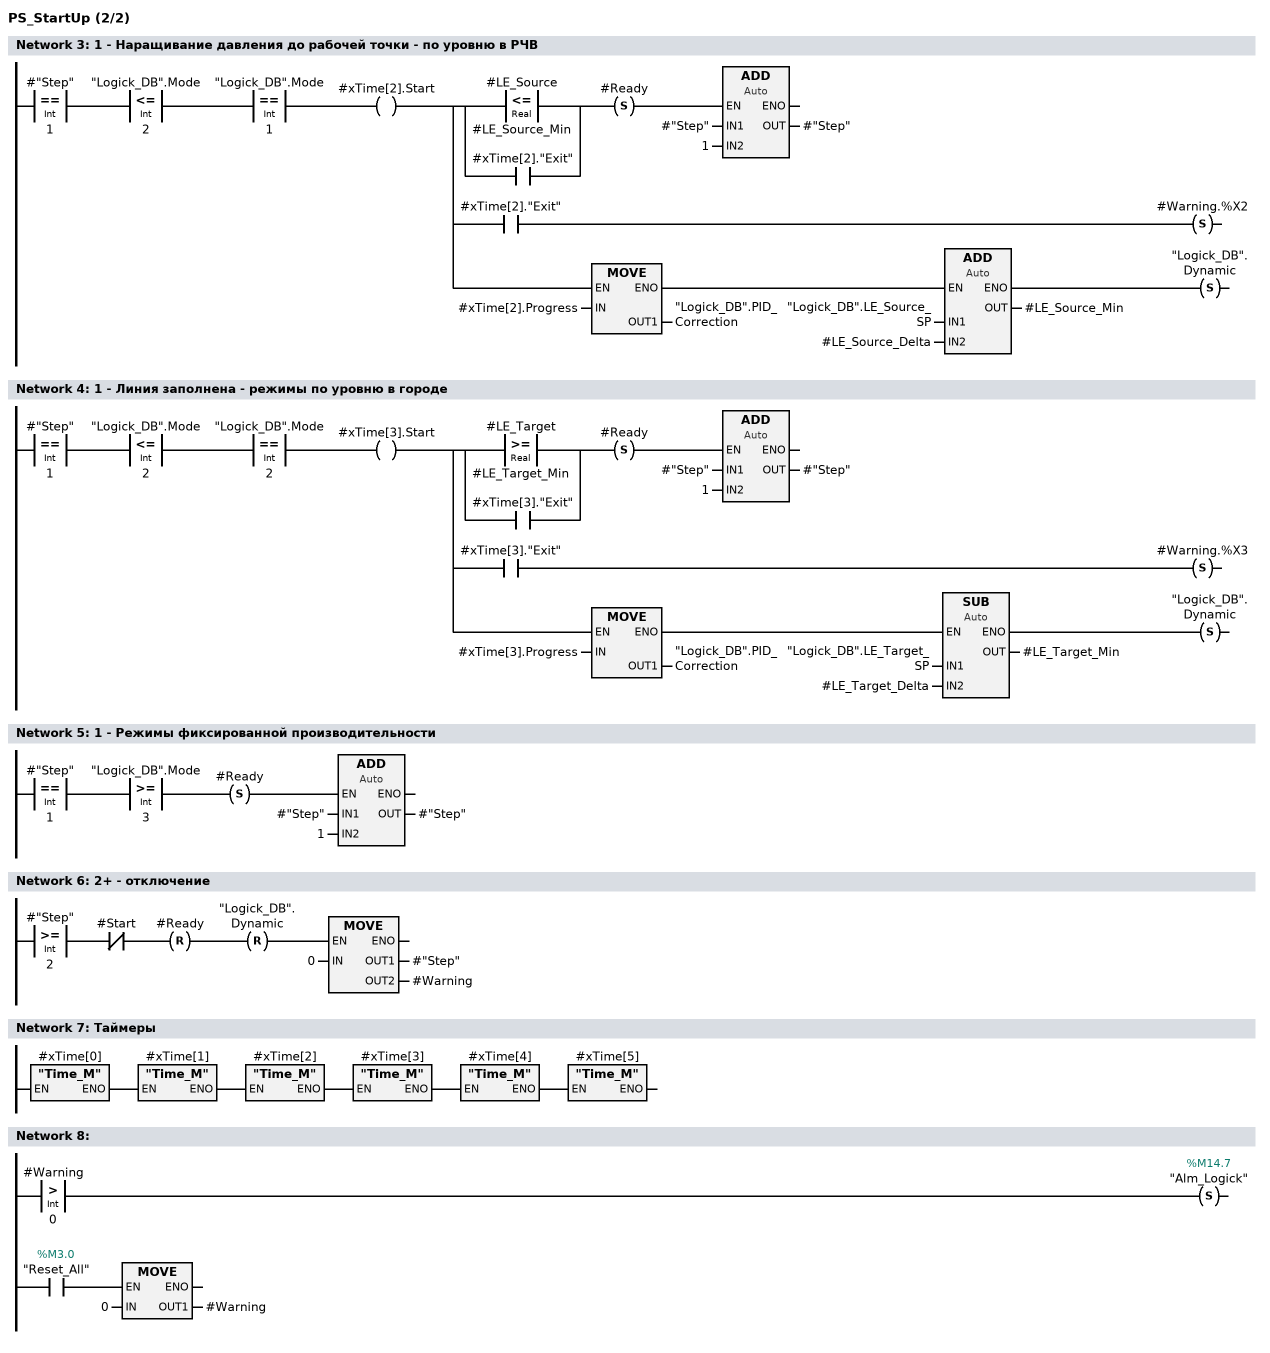
   RUNG wire#powerrail
      { S7_Templates := "SrcType := Int" } EQ_Contact(in1 := #"Step", in2 := 1)
      { S7_Templates := "SrcType := Int" } LE_Contact(in1 := "Logick_DB".Mode, in2 := 2)
      { S7_Templates := "SrcType := Int" } EQ_Contact(in1 := "Logick_DB".Mode, in2 := 1)
      Coil( #xTime[2].Start )
      wire#w1
      { S7_Templates := "SrcType := Real" } LE_Contact(in1 := #LE_Source, in2 := #LE_Source_Min)
      wire#w2
      S_Coil( #Ready )
      Add(in1 := #"Step", in2 := 1, out => #"Step")
   END_RUNG
   RUNG wire#w1
      Contact( #xTime[2]."Exit" )
   END_RUNG wire#w2
   RUNG wire#w1
      Contact( #xTime[2]."Exit" )
      S_Coil( #Warning.%X2 )
   END_RUNG
   RUNG wire#w1
      Move(in := #xTime[2].Progress, out1 => "Logick_DB".PID_Correction)
      Add(in1 := "Logick_DB".LE_Source_SP, in2 := #LE_Source_Delta, out => #LE_Source_Min)
      S_Coil( "Logick_DB".Dynamic )
   END_RUNG
   // the same network as SCL:
   #xTime[2].Start := (#"Step" = 1) AND ("Logick_DB".Mode <= 2) AND ("Logick_DB".Mode = 1);
   #_w1 := (#"Step" = 1) AND ("Logick_DB".Mode <= 2) AND ("Logick_DB".Mode = 1);
   IF #_w1 AND ((#LE_Source <= #LE_Source_Min) OR #xTime[2]."Exit") THEN
       #Ready := TRUE;
       #"Step" := #"Step" + 1;
   END_IF;
   IF #_w1 AND #xTime[2]."Exit" THEN #Warning.%X2 := TRUE; END_IF;
   IF #_w1 THEN
       "Logick_DB".PID_Correction := #xTime[2].Progress;
       #LE_Source_Min := "Logick_DB".LE_Source_SP + #LE_Source_Delta;
       "Logick_DB".Dynamic := TRUE;
   END_IF;
END_REGION

REGION Network 4: 1 - Линия заполнена - режимы по уровню в городе
   RUNG wire#powerrail
      { S7_Templates := "SrcType := Int" } EQ_Contact(in1 := #"Step", in2 := 1)
      { S7_Templates := "SrcType := Int" } LE_Contact(in1 := "Logick_DB".Mode, in2 := 2)
      { S7_Templates := "SrcType := Int" } EQ_Contact(in1 := "Logick_DB".Mode, in2 := 2)
      Coil( #xTime[3].Start )
      wire#w1
      { S7_Templates := "SrcType := Real" } GE_Contact(in1 := #LE_Target, in2 := #LE_Target_Min)
      wire#w2
      S_Coil( #Ready )
      Add(in1 := #"Step", in2 := 1, out => #"Step")
   END_RUNG
   RUNG wire#w1
      Contact( #xTime[3]."Exit" )
   END_RUNG wire#w2
   RUNG wire#w1
      Contact( #xTime[3]."Exit" )
      S_Coil( #Warning.%X3 )
   END_RUNG
   RUNG wire#w1
      Move(in := #xTime[3].Progress, out1 => "Logick_DB".PID_Correction)
      Sub(in1 := "Logick_DB".LE_Target_SP, in2 := #LE_Target_Delta, out => #LE_Target_Min)
      S_Coil( "Logick_DB".Dynamic )
   END_RUNG
   // the same network as SCL:
   #xTime[3].Start := (#"Step" = 1) AND ("Logick_DB".Mode <= 2) AND ("Logick_DB".Mode = 2);
   #_w1 := (#"Step" = 1) AND ("Logick_DB".Mode <= 2) AND ("Logick_DB".Mode = 2);
   IF #_w1 AND ((#LE_Target >= #LE_Target_Min) OR #xTime[3]."Exit") THEN
       #Ready := TRUE;
       #"Step" := #"Step" + 1;
   END_IF;
   IF #_w1 AND #xTime[3]."Exit" THEN #Warning.%X3 := TRUE; END_IF;
   IF #_w1 THEN
       "Logick_DB".PID_Correction := #xTime[3].Progress;
       #LE_Target_Min := "Logick_DB".LE_Target_SP - #LE_Target_Delta;
       "Logick_DB".Dynamic := TRUE;
   END_IF;
END_REGION

REGION Network 5: 1 - Режимы фиксированной производительности
   RUNG wire#powerrail
      { S7_Templates := "SrcType := Int" } EQ_Contact(in1 := #"Step", in2 := 1)
      { S7_Templates := "SrcType := Int" } GE_Contact(in1 := "Logick_DB".Mode, in2 := 3)
      S_Coil( #Ready )
      Add(in1 := #"Step", in2 := 1, out => #"Step")
   END_RUNG
   // the same network as SCL:
   IF (#"Step" = 1) AND ("Logick_DB".Mode >= 3) THEN
       #Ready := TRUE;
       #"Step" := #"Step" + 1;
   END_IF;
END_REGION

REGION Network 6: 2+ - отключение
   RUNG wire#powerrail
      { S7_Templates := "SrcType := Int" } GE_Contact(in1 := #"Step", in2 := 2)
      I_Contact( #Start )
      R_Coil( #Ready )
      R_Coil( "Logick_DB".Dynamic )
      Move(in := 0, out1 => #"Step", out2 => #Warning)
   END_RUNG
   // the same network as SCL:
   IF (#"Step" >= 2) AND NOT #Start THEN
       #Ready := FALSE;
       "Logick_DB".Dynamic := FALSE;
       #"Step" := 0;
       #Warning := 0;
   END_IF;
END_REGION

REGION Network 7: Таймеры
   RUNG wire#powerrail
      #xTime[0]()
      #xTime[1]()
      #xTime[2]()
      #xTime[3]()
      #xTime[4]()
      #xTime[5]()
   END_RUNG
   // the same network as SCL:
   #xTime[0](ENO => #_w1);   // "Time_M"
   #xTime[1](EN := #_w1, ENO => #_w2);   // "Time_M"
   #xTime[2](EN := #_w2, ENO => #_w3);   // "Time_M"
   #xTime[3](EN := #_w3, ENO => #_w4);   // "Time_M"
   #xTime[4](EN := #_w4, ENO => #_w5);   // "Time_M"
   IF #_w5 THEN
       #xTime[5]();   // "Time_M"
   END_IF;
END_REGION

REGION Network 8
   RUNG wire#powerrail
      { S7_Templates := "SrcType := Int" } GT_Contact(in1 := #Warning, in2 := 0)
      S_Coil( "Alm_Logick" )
   END_RUNG
   RUNG wire#powerrail
      Contact( "Reset_All" )
      Move(in := 0, out1 => #Warning)
   END_RUNG
   // the same network as SCL:
   IF #Warning > 0 THEN "Alm_Logick" := TRUE; END_IF;
   IF "Reset_All" THEN #Warning := 0; END_IF;
END_REGION
END_FUNCTION_BLOCK

FUNCTION_BLOCK "Time_M"   // FB92, LAD
{ S7_Optimized_Access := 'FALSE' }
VERSION : 0.1
// stored: AutoNumber false, IsIECCheckEnabled false, SetENOAutomatically false, UDAEnableTagReadback false
   VAR DB_SPECIFIC
      SP_M { S7_SetPoint := 'True'} : Int;
      SP_S { S7_SetPoint := 'True'} : Int := 30;
      Now_M : Int;
      Now_S : Int;
      Rev_M : Int;
      Rev_S : Int;
      Progress : Real;
      Start : Bool;
      "Exit" : Bool;
      Pause : Bool;
      Reset : Bool;
   END_VAR
   VAR_TEMP
      Full_SP_S : Int;
      Full_Now_S : Int;
      Full_Delta_S : Int;
   END_VAR
   VAR_TEMP   // added for the SCL form of the ladder/FBD networks
      _w1 : Bool;
   END_VAR
BEGIN

REGION Network 1: Подсчёт времени
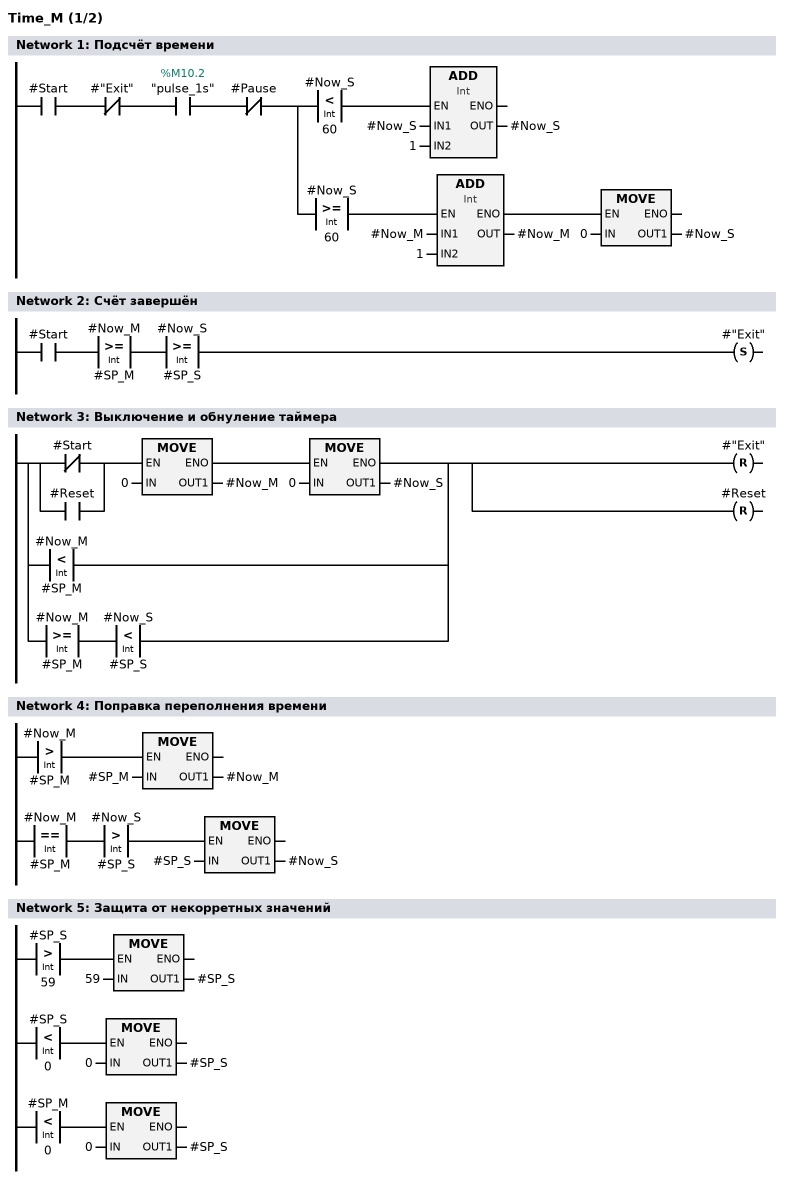
   RUNG wire#powerrail
      Contact( #Start )
      I_Contact( #"Exit" )
      Contact( "pulse_1s" )
      I_Contact( #Pause )
      wire#w1
      { S7_Templates := "SrcType := Int" } LT_Contact(in1 := #Now_S, in2 := 60)
      { S7_Templates := "SrcType := Int"; S7_GenerateENO := "TRUE" } Add(in1 := #Now_S, in2 := 1, out => #Now_S)
   END_RUNG
   RUNG wire#w1
      { S7_Templates := "SrcType := Int" } GE_Contact(in1 := #Now_S, in2 := 60)
      { S7_Templates := "SrcType := Int"; S7_GenerateENO := "TRUE" } Add(in1 := #Now_M, in2 := 1, out => #Now_M)
      { S7_GenerateENO := "TRUE" } Move(in := 0, out1 => #Now_S)
   END_RUNG
   // the same network as SCL:
   // ENO of a box is taken as its EN; it also drops when the box reports an error
   #_w1 := #Start AND NOT #"Exit" AND "pulse_1s" AND NOT #Pause;
   IF #_w1 AND (#Now_S < 60) THEN #Now_S := #Now_S + 1; END_IF;
   IF #_w1 AND (#Now_S >= 60) THEN
       #Now_M := #Now_M + 1;
       #Now_S := 0;
   END_IF;
END_REGION

REGION Network 2: Счёт завершён
   RUNG wire#powerrail
      Contact( #Start )
      { S7_Templates := "SrcType := Int" } GE_Contact(in1 := #Now_M, in2 := #SP_M)
      { S7_Templates := "SrcType := Int" } GE_Contact(in1 := #Now_S, in2 := #SP_S)
      S_Coil( #"Exit" )
   END_RUNG
   // the same network as SCL:
   IF #Start AND (#Now_M >= #SP_M) AND (#Now_S >= #SP_S) THEN #"Exit" := TRUE; END_IF;
END_REGION

REGION Network 3: Выключение и обнуление таймера
   RUNG wire#powerrail
      I_Contact( #Start )
      wire#w1
      { S7_GenerateENO := "TRUE" } Move(in := 0, out1 => #Now_M)
      { S7_GenerateENO := "TRUE" } Move(in := 0, out1 => #Now_S)
      wire#w2
      R_Coil( #"Exit" )
   END_RUNG
   RUNG wire#powerrail
      Contact( #Reset )
   END_RUNG wire#w1
   RUNG wire#powerrail
      { S7_Templates := "SrcType := Int" } LT_Contact(in1 := #Now_M, in2 := #SP_M)
   END_RUNG wire#w2
   RUNG wire#powerrail
      { S7_Templates := "SrcType := Int" } GE_Contact(in1 := #Now_M, in2 := #SP_M)
      { S7_Templates := "SrcType := Int" } LT_Contact(in1 := #Now_S, in2 := #SP_S)
   END_RUNG wire#w2
   RUNG wire#w2
      R_Coil( #Reset )
   END_RUNG
   // the same network as SCL:
   // ENO of a box is taken as its EN; it also drops when the box reports an error
   #_w1 := NOT #Start OR #Reset;
   IF #_w1 THEN
       #Now_M := 0;
       #Now_S := 0;
   END_IF;
   IF #_w1 OR (#Now_M < #SP_M) OR ((#Now_M >= #SP_M) AND (#Now_S < #SP_S)) THEN
       #"Exit" := FALSE;
       #Reset := FALSE;
   END_IF;
END_REGION

REGION Network 4: Поправка переполнения времени
   RUNG wire#powerrail
      { S7_Templates := "SrcType := Int" } GT_Contact(in1 := #Now_M, in2 := #SP_M)
      { S7_GenerateENO := "TRUE" } Move(in := #SP_M, out1 => #Now_M)
   END_RUNG
   RUNG wire#powerrail
      { S7_Templates := "SrcType := Int" } EQ_Contact(in1 := #Now_M, in2 := #SP_M)
      { S7_Templates := "SrcType := Int" } GT_Contact(in1 := #Now_S, in2 := #SP_S)
      { S7_GenerateENO := "TRUE" } Move(in := #SP_S, out1 => #Now_S)
   END_RUNG
   // the same network as SCL:
   IF #Now_M > #SP_M THEN #Now_M := #SP_M; END_IF;
   IF (#Now_M = #SP_M) AND (#Now_S > #SP_S) THEN #Now_S := #SP_S; END_IF;
END_REGION

REGION Network 5: Защита от некорретных значений
   RUNG wire#powerrail
      { S7_Templates := "SrcType := Int" } GT_Contact(in1 := #SP_S, in2 := 59)
      { S7_GenerateENO := "TRUE" } Move(in := 59, out1 => #SP_S)
   END_RUNG
   RUNG wire#powerrail
      { S7_Templates := "SrcType := Int" } LT_Contact(in1 := #SP_S, in2 := 0)
      { S7_GenerateENO := "TRUE" } Move(in := 0, out1 => #SP_S)
   END_RUNG
   RUNG wire#powerrail
      { S7_Templates := "SrcType := Int" } LT_Contact(in1 := #SP_M, in2 := 0)
      { S7_GenerateENO := "TRUE" } Move(in := 0, out1 => #SP_S)
   END_RUNG
   // the same network as SCL:
   IF #SP_S > 59 THEN #SP_S := 59; END_IF;
   IF #SP_S < 0 THEN #SP_S := 0; END_IF;
   IF #SP_M < 0 THEN #SP_S := 0; END_IF;
END_REGION

REGION Network 6: Обратный отсчёт
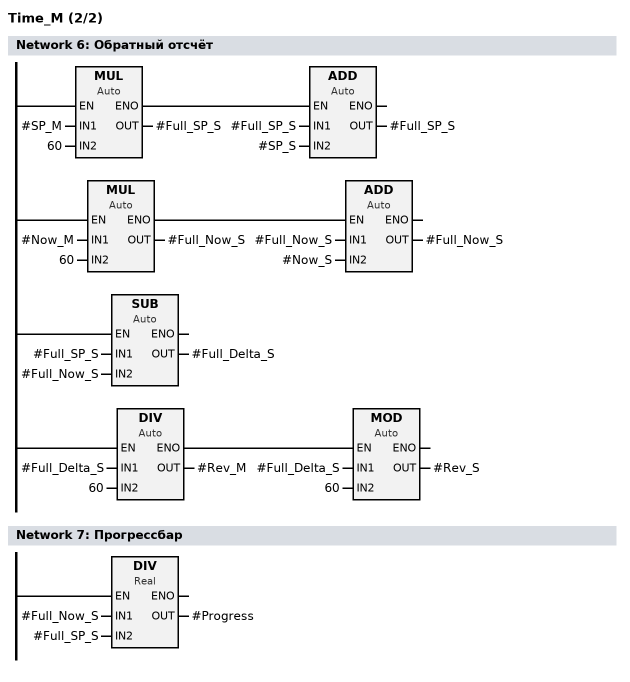
   RUNG wire#powerrail
      Mul(in1 := #SP_M, in2 := 60, out => #Full_SP_S)
      Add(in1 := #Full_SP_S, in2 := #SP_S, out => #Full_SP_S)
   END_RUNG
   RUNG wire#powerrail
      Mul(in1 := #Now_M, in2 := 60, out => #Full_Now_S)
      Add(in1 := #Full_Now_S, in2 := #Now_S, out => #Full_Now_S)
   END_RUNG
   RUNG wire#powerrail
      Sub(in1 := #Full_SP_S, in2 := #Full_Now_S, out => #Full_Delta_S)
   END_RUNG
   RUNG wire#powerrail
      Div(in1 := #Full_Delta_S, in2 := 60, out => #Rev_M)
      Mod(in1 := #Full_Delta_S, in2 := 60, out => #Rev_S)
   END_RUNG
   // the same network as SCL:
   #Full_SP_S := #SP_M * 60;
   #Full_SP_S := #Full_SP_S + #SP_S;
   #Full_Now_S := #Now_M * 60;
   #Full_Now_S := #Full_Now_S + #Now_S;
   #Full_Delta_S := #Full_SP_S - #Full_Now_S;
   #Rev_M := #Full_Delta_S / 60;
   #Rev_S := #Full_Delta_S MOD 60;
END_REGION

REGION Network 7: Прогрессбар
   RUNG wire#powerrail
      { S7_Templates := "SrcType := Real" } Div(in1 := #Full_Now_S, in2 := #Full_SP_S, out => #Progress)
   END_RUNG
   // the same network as SCL:
   #Progress := #Full_Now_S / #Full_SP_S;
END_REGION
END_FUNCTION_BLOCK

FUNCTION_BLOCK "PS_cnt"   // FB12, LAD
{ S7_Optimized_Access := 'FALSE' }
VERSION : 0.1
// stored: AutoNumber false, IsIECCheckEnabled false, SetENOAutomatically false, UDAEnableTagReadback false
   VAR_INPUT
      SP : Real;
      REQ : Int;
   END_VAR
   VAR_IN_OUT
      cnt : Int;   // Число насосов в работе
   END_VAR
   VAR DB_SPECIFIC
      Select_CMD : Bool;   // Запрос выбора насоса
      Select_Mode : Bool;   // 0 - для останова, 1 - для запуска
      Select_PS : Int;   // Выбранный насос
      PS_Add_Ready : Bool;   // Насосы вышли на общую точку
      PS_Add_CMD : Bool;   // Запрос выхода на общую точку
      SP_Low : Real := 40.0;   // Нижняя рабочая точка
      SP_High { S7_SetPoint := 'True'} : Real := 45.0;   // Верхняя рабочая точка
      SP_Min { S7_SetPoint := 'True'} : Real := 36.0;   // Точка открытия обратного клапана
      cnt_delta { S7_SetPoint := 'True'} : Real := 0.5;   // Смещение точки открытия обратного клапана на 1 работающий насос
      "Step" : Int;
      REQ_cnt : Int;
      PS_R_OFF : Int;   // Насос для отключения при ротации
      PS_R_ON : Int;   // Насос для запуска при ротации
      pos : Array[0..15] of Bool;
      tmp : Array[0..15] of Real;
   END_VAR
   VAR
      T_Delay_ON { S7_SetPoint := 'True'} : "Time_M";   // Задержка запуска след. насоса
      T_Delay_OFF { S7_SetPoint := 'True'} : "Time_M";   // Задержка останова след. насоса
   END_VAR
   VAR_TEMP
      x_delta : Real;
   END_VAR
   VAR_TEMP   // added for the SCL form of the ladder/FBD networks
      _w1 : Bool;
      _w2 : Bool;
      _w3 : Bool;
      _w4 : Bool;
      _w5 : Bool;
      _w6 : Bool;
      _w7 : Bool;
      _w8 : Bool;
   END_VAR
BEGIN

REGION Network 1: Коррекция нижней рабочей точки по числу насосов
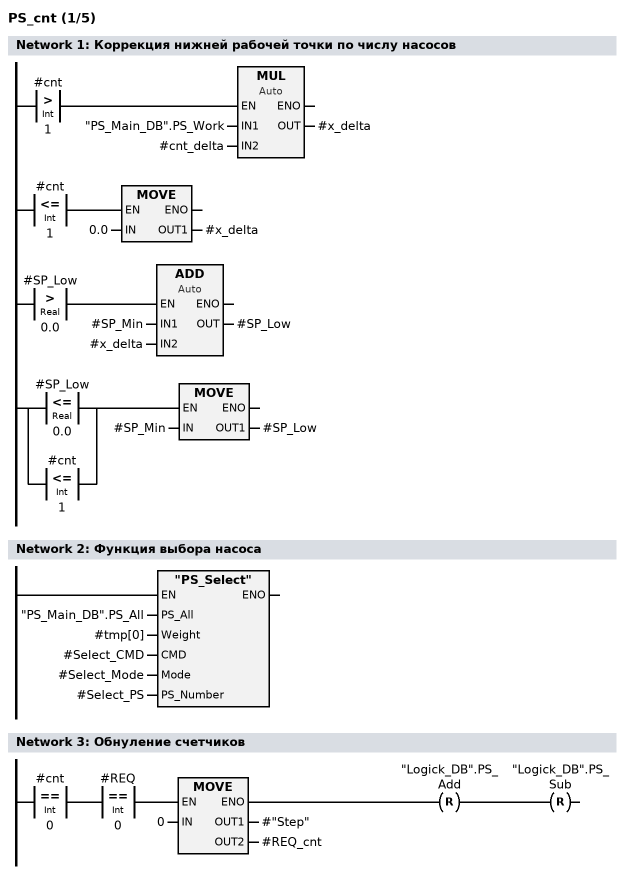
   RUNG wire#powerrail
      { S7_Templates := "SrcType := Int" } GT_Contact(in1 := #cnt, in2 := 1)
      Mul(in1 := "PS_Main_DB".PS_Work, in2 := #cnt_delta, out => #x_delta)
   END_RUNG
   RUNG wire#powerrail
      { S7_Templates := "SrcType := Int" } LE_Contact(in1 := #cnt, in2 := 1)
      Move(in := 0.0, out1 => #x_delta)
   END_RUNG
   RUNG wire#powerrail
      { S7_Templates := "SrcType := Real" } GT_Contact(in1 := #SP_Low, in2 := 0.0)
      Add(in1 := #SP_Min, in2 := #x_delta, out => #SP_Low)
   END_RUNG
   RUNG wire#powerrail
      { S7_Templates := "SrcType := Real" } LE_Contact(in1 := #SP_Low, in2 := 0.0)
      wire#w1
      Move(in := #SP_Min, out1 => #SP_Low)
   END_RUNG
   RUNG wire#powerrail
      { S7_Templates := "SrcType := Int" } LE_Contact(in1 := #cnt, in2 := 1)
   END_RUNG wire#w1
   // the same network as SCL:
   IF #cnt > 1 THEN #x_delta := "PS_Main_DB".PS_Work * #cnt_delta; END_IF;
   IF #cnt <= 1 THEN #x_delta := 0.0; END_IF;
   IF #SP_Low > 0.0 THEN #SP_Low := #SP_Min + #x_delta; END_IF;
   IF (#SP_Low <= 0.0) OR (#cnt <= 1) THEN #SP_Low := #SP_Min; END_IF;
END_REGION

REGION Network 2: Функция выбора насоса
   RUNG wire#powerrail
      "PS_Select"(PS_All := "PS_Main_DB".PS_All, Weight := #tmp[0], CMD := #Select_CMD, Mode := #Select_Mode, PS_Number := #Select_PS)
   END_RUNG
   // the same network as SCL:
   "PS_Select"(PS_All := "PS_Main_DB".PS_All,
               Weight := #tmp[0],
               CMD := #Select_CMD,
               Mode := #Select_Mode,
               PS_Number := #Select_PS);
END_REGION

REGION Network 3: Обнуление счетчиков
   RUNG wire#powerrail
      { S7_Templates := "SrcType := Int" } EQ_Contact(in1 := #cnt, in2 := 0)
      { S7_Templates := "SrcType := Int" } EQ_Contact(in1 := #REQ, in2 := 0)
      Move(in := 0, out1 => #"Step", out2 => #REQ_cnt)
      R_Coil( "Logick_DB".PS_Add )
      R_Coil( "Logick_DB".PS_Sub )
   END_RUNG
   // the same network as SCL:
   IF (#cnt = 0) AND (#REQ = 0) THEN
       #"Step" := 0;
       #REQ_cnt := 0;
       "Logick_DB".PS_Add := FALSE;
       "Logick_DB".PS_Sub := FALSE;
   END_IF;
END_REGION

REGION Network 4: Запуск первого насоса
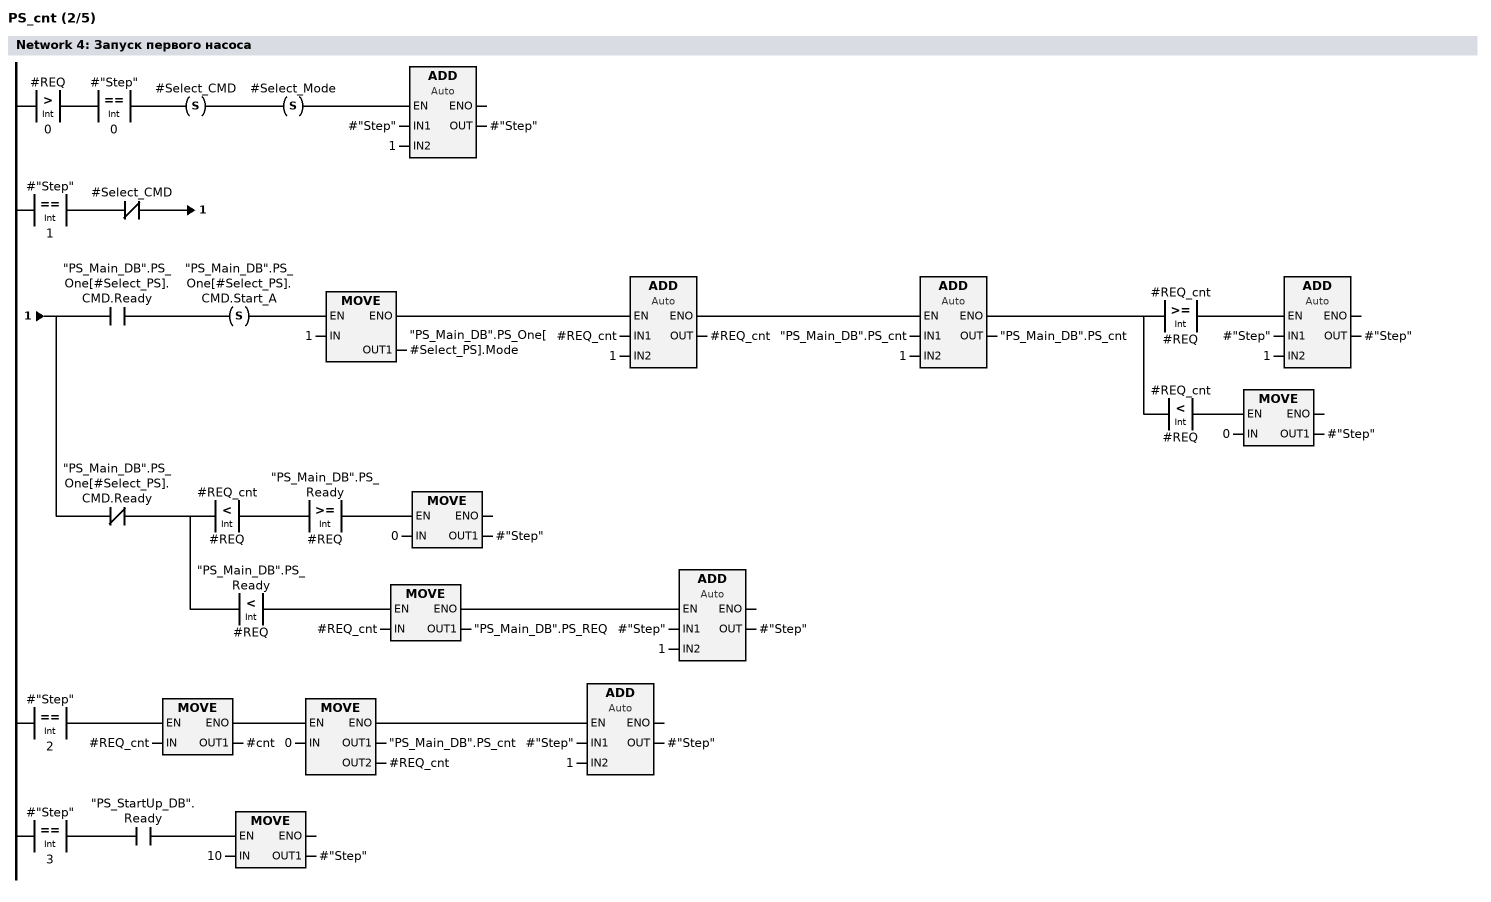
   RUNG wire#powerrail
      { S7_Templates := "SrcType := Int" } GT_Contact(in1 := #REQ, in2 := 0)
      { S7_Templates := "SrcType := Int" } EQ_Contact(in1 := #"Step", in2 := 0)
      S_Coil( #Select_CMD )
      S_Coil( #Select_Mode )
      Add(in1 := #"Step", in2 := 1, out => #"Step")
   END_RUNG
   RUNG wire#powerrail
      { S7_Templates := "SrcType := Int" } EQ_Contact(in1 := #"Step", in2 := 1)
      I_Contact( #Select_CMD )
      wire#w1
      Contact( "PS_Main_DB".PS_One[#Select_PS].CMD.Ready )
      S_Coil( "PS_Main_DB".PS_One[#Select_PS].CMD.Start_A )
      Move(in := 1, out1 => "PS_Main_DB".PS_One[#Select_PS].Mode)
      Add(in1 := #REQ_cnt, in2 := 1, out => #REQ_cnt)
      Add(in1 := "PS_Main_DB".PS_cnt, in2 := 1, out => "PS_Main_DB".PS_cnt)
      wire#w2
      { S7_Templates := "SrcType := Int" } GE_Contact(in1 := #REQ_cnt, in2 := #REQ)
      Add(in1 := #"Step", in2 := 1, out => #"Step")
   END_RUNG
   RUNG wire#w2
      { S7_Templates := "SrcType := Int" } LT_Contact(in1 := #REQ_cnt, in2 := #REQ)
      Move(in := 0, out1 => #"Step")
   END_RUNG
   RUNG wire#w1
      I_Contact( "PS_Main_DB".PS_One[#Select_PS].CMD.Ready )
      wire#w3
      { S7_Templates := "SrcType := Int" } LT_Contact(in1 := #REQ_cnt, in2 := #REQ)
      { S7_Templates := "SrcType := Int" } GE_Contact(in1 := "PS_Main_DB".PS_Ready, in2 := #REQ)
      Move(in := 0, out1 => #"Step")
   END_RUNG
   RUNG wire#w3
      { S7_Templates := "SrcType := Int" } LT_Contact(in1 := "PS_Main_DB".PS_Ready, in2 := #REQ)
      Move(in := #REQ_cnt, out1 => "PS_Main_DB".PS_REQ)
      Add(in1 := #"Step", in2 := 1, out => #"Step")
   END_RUNG
   RUNG wire#powerrail
      { S7_Templates := "SrcType := Int" } EQ_Contact(in1 := #"Step", in2 := 2)
      Move(in := #REQ_cnt, out1 => #cnt)
      Move(in := 0, out1 => "PS_Main_DB".PS_cnt, out2 => #REQ_cnt)
      Add(in1 := #"Step", in2 := 1, out => #"Step")
   END_RUNG
   RUNG wire#powerrail
      { S7_Templates := "SrcType := Int" } EQ_Contact(in1 := #"Step", in2 := 3)
      Contact( "PS_StartUp_DB".Ready )
      Move(in := 10, out1 => #"Step")
   END_RUNG
   // the same network as SCL:
   IF (#REQ > 0) AND (#"Step" = 0) THEN
       #Select_CMD := TRUE;
       #Select_Mode := TRUE;
       #"Step" := #"Step" + 1;
   END_IF;
   #_w1 := (#"Step" = 1) AND NOT #Select_CMD;
   #_w2 := #_w1 AND "PS_Main_DB".PS_One[#Select_PS].CMD.Ready;
   IF #_w2 THEN
       "PS_Main_DB".PS_One[#Select_PS].CMD.Start_A := TRUE;
       "PS_Main_DB".PS_One[#Select_PS].Mode := 1;
       #REQ_cnt := #REQ_cnt + 1;
       "PS_Main_DB".PS_cnt := "PS_Main_DB".PS_cnt + 1;
   END_IF;
   IF #_w2 AND (#REQ_cnt >= #REQ) THEN #"Step" := #"Step" + 1; END_IF;
   IF #_w2 AND (#REQ_cnt < #REQ) THEN #"Step" := 0; END_IF;
   #_w3 := #_w1 AND NOT "PS_Main_DB".PS_One[#Select_PS].CMD.Ready;
   IF #_w3 AND (#REQ_cnt < #REQ) AND ("PS_Main_DB".PS_Ready >= #REQ) THEN #"Step" := 0; END_IF;
   IF #_w3 AND ("PS_Main_DB".PS_Ready < #REQ) THEN
       "PS_Main_DB".PS_REQ := #REQ_cnt;
       #"Step" := #"Step" + 1;
   END_IF;
   IF #"Step" = 2 THEN
       #cnt := #REQ_cnt;
       "PS_Main_DB".PS_cnt := 0;
       #REQ_cnt := 0;
       #"Step" := #"Step" + 1;
   END_IF;
   IF (#"Step" = 3) AND "PS_StartUp_DB".Ready THEN #"Step" := 10; END_IF;
END_REGION

REGION Network 5: Добавление нового насоса
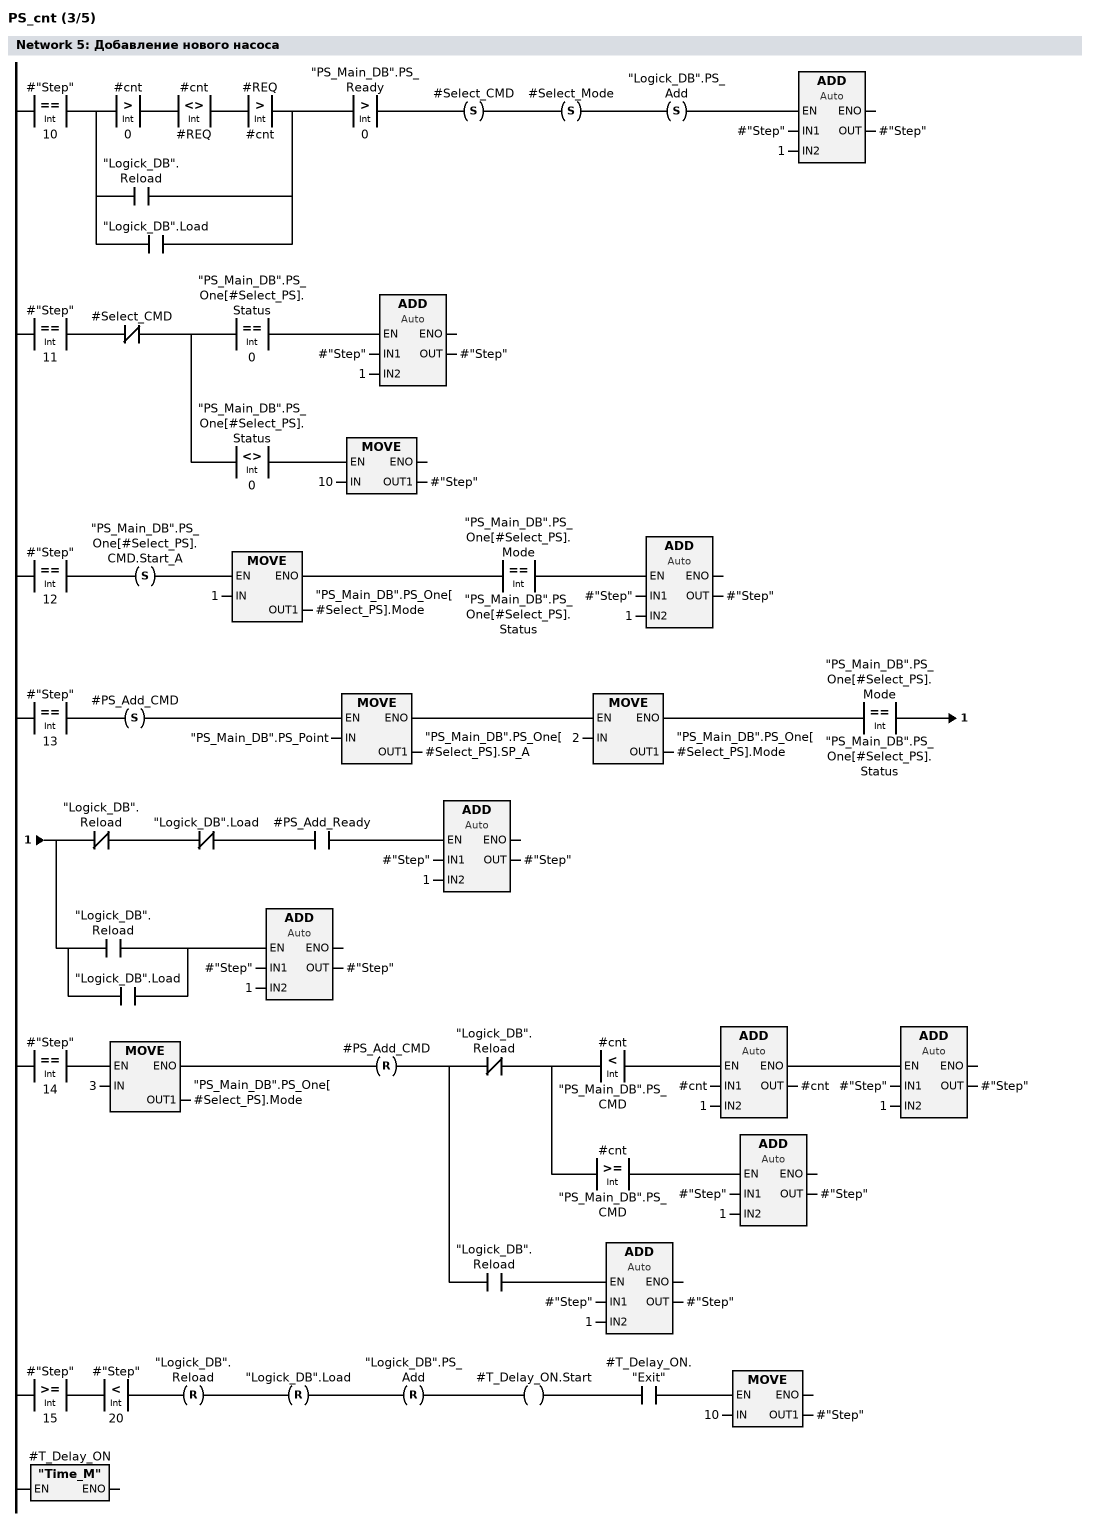
   RUNG wire#powerrail
      { S7_Templates := "SrcType := Int" } EQ_Contact(in1 := #"Step", in2 := 10)
      wire#w1
      { S7_Templates := "SrcType := Int" } GT_Contact(in1 := #cnt, in2 := 0)
      { S7_Templates := "SrcType := Int" } NE_Contact(in1 := #cnt, in2 := #REQ)
      { S7_Templates := "SrcType := Int" } GT_Contact(in1 := #REQ, in2 := #cnt)
      wire#w2
      { S7_Templates := "SrcType := Int" } GT_Contact(in1 := "PS_Main_DB".PS_Ready, in2 := 0)
      S_Coil( #Select_CMD )
      S_Coil( #Select_Mode )
      S_Coil( "Logick_DB".PS_Add )
      Add(in1 := #"Step", in2 := 1, out => #"Step")
   END_RUNG
   RUNG wire#w1
      Contact( "Logick_DB".Reload )
   END_RUNG wire#w2
   RUNG wire#w1
      Contact( "Logick_DB".Load )
   END_RUNG wire#w2
   RUNG wire#powerrail
      { S7_Templates := "SrcType := Int" } EQ_Contact(in1 := #"Step", in2 := 11)
      I_Contact( #Select_CMD )
      wire#w3
      { S7_Templates := "SrcType := Int" } EQ_Contact(in1 := "PS_Main_DB".PS_One[#Select_PS].Status, in2 := 0)
      Add(in1 := #"Step", in2 := 1, out => #"Step")
   END_RUNG
   RUNG wire#w3
      { S7_Templates := "SrcType := Int" } NE_Contact(in1 := "PS_Main_DB".PS_One[#Select_PS].Status, in2 := 0)
      Move(in := 10, out1 => #"Step")
   END_RUNG
   RUNG wire#powerrail
      { S7_Templates := "SrcType := Int" } EQ_Contact(in1 := #"Step", in2 := 12)
      S_Coil( "PS_Main_DB".PS_One[#Select_PS].CMD.Start_A )
      Move(in := 1, out1 => "PS_Main_DB".PS_One[#Select_PS].Mode)
      { S7_Templates := "SrcType := Int" } EQ_Contact(in1 := "PS_Main_DB".PS_One[#Select_PS].Mode, in2 := "PS_Main_DB".PS_One[#Select_PS].Status)
      Add(in1 := #"Step", in2 := 1, out => #"Step")
   END_RUNG
   RUNG wire#powerrail
      { S7_Templates := "SrcType := Int" } EQ_Contact(in1 := #"Step", in2 := 13)
      S_Coil( #PS_Add_CMD )
      Move(in := "PS_Main_DB".PS_Point, out1 => "PS_Main_DB".PS_One[#Select_PS].SP_A)
      Move(in := 2, out1 => "PS_Main_DB".PS_One[#Select_PS].Mode)
      { S7_Templates := "SrcType := Int" } EQ_Contact(in1 := "PS_Main_DB".PS_One[#Select_PS].Mode, in2 := "PS_Main_DB".PS_One[#Select_PS].Status)
      wire#w4
      I_Contact( "Logick_DB".Reload )
      I_Contact( "Logick_DB".Load )
      Contact( #PS_Add_Ready )
      Add(in1 := #"Step", in2 := 1, out => #"Step")
   END_RUNG
   RUNG wire#w4
      Contact( "Logick_DB".Reload )
      wire#w5
      Add(in1 := #"Step", in2 := 1, out => #"Step")
   END_RUNG
   RUNG wire#w4
      Contact( "Logick_DB".Load )
   END_RUNG wire#w5
   RUNG wire#powerrail
      { S7_Templates := "SrcType := Int" } EQ_Contact(in1 := #"Step", in2 := 14)
      Move(in := 3, out1 => "PS_Main_DB".PS_One[#Select_PS].Mode)
      R_Coil( #PS_Add_CMD )
      wire#w6
      I_Contact( "Logick_DB".Reload )
      wire#w7
      { S7_Templates := "SrcType := Int" } LT_Contact(in1 := #cnt, in2 := "PS_Main_DB".PS_CMD)
      Add(in1 := #cnt, in2 := 1, out => #cnt)
      Add(in1 := #"Step", in2 := 1, out => #"Step")
   END_RUNG
   RUNG wire#w7
      { S7_Templates := "SrcType := Int" } GE_Contact(in1 := #cnt, in2 := "PS_Main_DB".PS_CMD)
      Add(in1 := #"Step", in2 := 1, out => #"Step")
   END_RUNG
   RUNG wire#w6
      Contact( "Logick_DB".Reload )
      Add(in1 := #"Step", in2 := 1, out => #"Step")
   END_RUNG
   RUNG wire#powerrail
      { S7_Templates := "SrcType := Int" } GE_Contact(in1 := #"Step", in2 := 15)
      { S7_Templates := "SrcType := Int" } LT_Contact(in1 := #"Step", in2 := 20)
      R_Coil( "Logick_DB".Reload )
      R_Coil( "Logick_DB".Load )
      R_Coil( "Logick_DB".PS_Add )
      Coil( #T_Delay_ON.Start )
      Contact( #T_Delay_ON."Exit" )
      Move(in := 10, out1 => #"Step")
   END_RUNG
   RUNG wire#powerrail
      #T_Delay_ON()
   END_RUNG
   // the same network as SCL:
   IF (#"Step" = 10) AND (((#cnt > 0) AND (#cnt <> #REQ) AND (#REQ > #cnt)) OR "Logick_DB".Reload OR "Logick_DB".Load) AND ("PS_Main_DB".PS_Ready > 0) THEN
       #Select_CMD := TRUE;
       #Select_Mode := TRUE;
       "Logick_DB".PS_Add := TRUE;
       #"Step" := #"Step" + 1;
   END_IF;
   #_w1 := (#"Step" = 11) AND NOT #Select_CMD;
   IF #_w1 AND ("PS_Main_DB".PS_One[#Select_PS].Status = 0) THEN #"Step" := #"Step" + 1; END_IF;
   IF #_w1 AND ("PS_Main_DB".PS_One[#Select_PS].Status <> 0) THEN #"Step" := 10; END_IF;
   #_w2 := #"Step" = 12;
   IF #_w2 THEN
       "PS_Main_DB".PS_One[#Select_PS].CMD.Start_A := TRUE;
       "PS_Main_DB".PS_One[#Select_PS].Mode := 1;
   END_IF;
   IF #_w2 AND ("PS_Main_DB".PS_One[#Select_PS].Mode = "PS_Main_DB".PS_One[#Select_PS].Status) THEN
       #"Step" := #"Step" + 1;
   END_IF;
   #_w3 := #"Step" = 13;
   IF #_w3 THEN
       #PS_Add_CMD := TRUE;
       "PS_Main_DB".PS_One[#Select_PS].SP_A := "PS_Main_DB".PS_Point;
       "PS_Main_DB".PS_One[#Select_PS].Mode := 2;
   END_IF;
   #_w4 := #_w3 AND ("PS_Main_DB".PS_One[#Select_PS].Mode = "PS_Main_DB".PS_One[#Select_PS].Status);
   IF #_w4 AND NOT "Logick_DB".Reload AND NOT "Logick_DB".Load AND #PS_Add_Ready THEN
       #"Step" := #"Step" + 1;
   END_IF;
   IF #_w4 AND ("Logick_DB".Reload OR "Logick_DB".Load) THEN #"Step" := #"Step" + 1; END_IF;
   #_w5 := #"Step" = 14;
   IF #_w5 THEN
       "PS_Main_DB".PS_One[#Select_PS].Mode := 3;
       #PS_Add_CMD := FALSE;
   END_IF;
   #_w6 := #_w5 AND NOT "Logick_DB".Reload;
   #_w7 := #_w6 AND (#cnt < "PS_Main_DB".PS_CMD);
   IF #_w7 THEN
       #cnt := #cnt + 1;
       #"Step" := #"Step" + 1;
   END_IF;
   IF #_w6 AND (#cnt >= "PS_Main_DB".PS_CMD) THEN #"Step" := #"Step" + 1; END_IF;
   IF #_w5 AND "Logick_DB".Reload THEN #"Step" := #"Step" + 1; END_IF;
   #_w8 := (#"Step" >= 15) AND (#"Step" < 20);
   IF #_w8 THEN
       "Logick_DB".Reload := FALSE;
       "Logick_DB".Load := FALSE;
       "Logick_DB".PS_Add := FALSE;
   END_IF;
   #T_Delay_ON.Start := #_w8;
   IF #_w8 AND #T_Delay_ON."Exit" THEN #"Step" := 10; END_IF;
   #T_Delay_ON();   // "Time_M"
END_REGION

REGION Network 6: Вывод из работы насоса
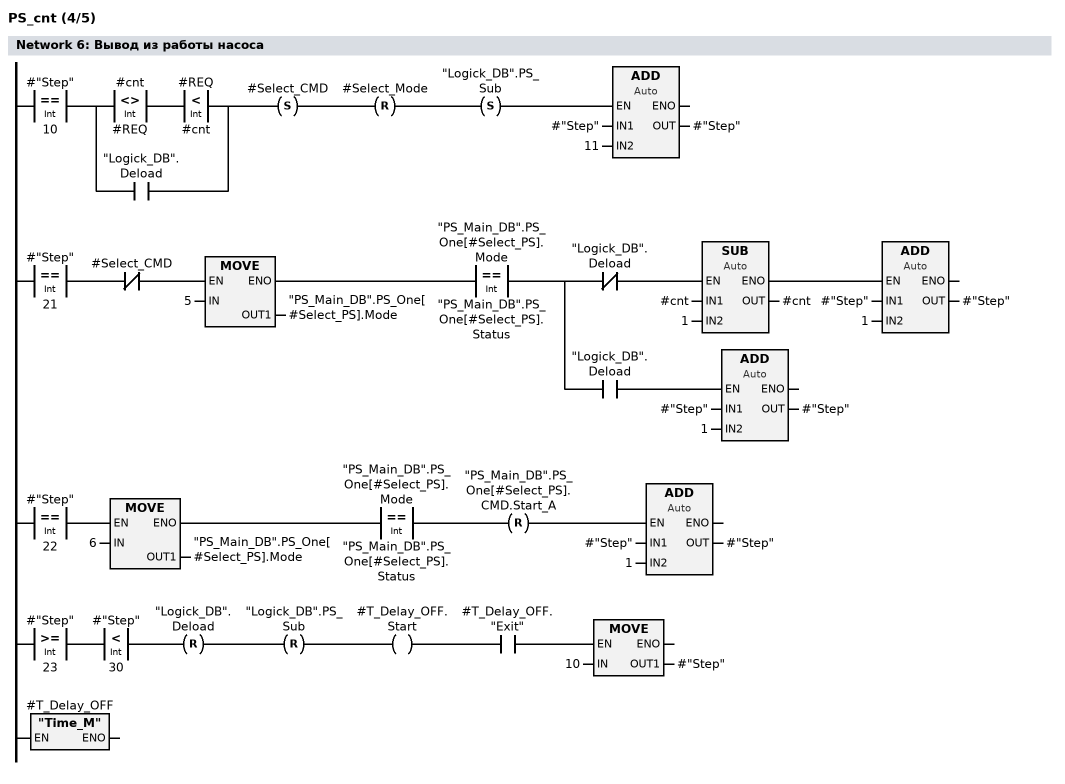
   RUNG wire#powerrail
      { S7_Templates := "SrcType := Int" } EQ_Contact(in1 := #"Step", in2 := 10)
      wire#w1
      { S7_Templates := "SrcType := Int" } NE_Contact(in1 := #cnt, in2 := #REQ)
      { S7_Templates := "SrcType := Int" } LT_Contact(in1 := #REQ, in2 := #cnt)
      wire#w2
      S_Coil( #Select_CMD )
      R_Coil( #Select_Mode )
      S_Coil( "Logick_DB".PS_Sub )
      Add(in1 := #"Step", in2 := 11, out => #"Step")
   END_RUNG
   RUNG wire#w1
      Contact( "Logick_DB".Deload )
   END_RUNG wire#w2
   RUNG wire#powerrail
      { S7_Templates := "SrcType := Int" } EQ_Contact(in1 := #"Step", in2 := 21)
      I_Contact( #Select_CMD )
      Move(in := 5, out1 => "PS_Main_DB".PS_One[#Select_PS].Mode)
      { S7_Templates := "SrcType := Int" } EQ_Contact(in1 := "PS_Main_DB".PS_One[#Select_PS].Mode, in2 := "PS_Main_DB".PS_One[#Select_PS].Status)
      wire#w3
      I_Contact( "Logick_DB".Deload )
      Sub(in1 := #cnt, in2 := 1, out => #cnt)
      Add(in1 := #"Step", in2 := 1, out => #"Step")
   END_RUNG
   RUNG wire#w3
      Contact( "Logick_DB".Deload )
      Add(in1 := #"Step", in2 := 1, out => #"Step")
   END_RUNG
   RUNG wire#powerrail
      { S7_Templates := "SrcType := Int" } EQ_Contact(in1 := #"Step", in2 := 22)
      Move(in := 6, out1 => "PS_Main_DB".PS_One[#Select_PS].Mode)
      { S7_Templates := "SrcType := Int" } EQ_Contact(in1 := "PS_Main_DB".PS_One[#Select_PS].Mode, in2 := "PS_Main_DB".PS_One[#Select_PS].Status)
      R_Coil( "PS_Main_DB".PS_One[#Select_PS].CMD.Start_A )
      Add(in1 := #"Step", in2 := 1, out => #"Step")
   END_RUNG
   RUNG wire#powerrail
      { S7_Templates := "SrcType := Int" } GE_Contact(in1 := #"Step", in2 := 23)
      { S7_Templates := "SrcType := Int" } LT_Contact(in1 := #"Step", in2 := 30)
      R_Coil( "Logick_DB".Deload )
      R_Coil( "Logick_DB".PS_Sub )
      Coil( #T_Delay_OFF.Start )
      Contact( #T_Delay_OFF."Exit" )
      Move(in := 10, out1 => #"Step")
   END_RUNG
   RUNG wire#powerrail
      #T_Delay_OFF()
   END_RUNG
   // the same network as SCL:
   IF (#"Step" = 10) AND (((#cnt <> #REQ) AND (#REQ < #cnt)) OR "Logick_DB".Deload) THEN
       #Select_CMD := TRUE;
       #Select_Mode := FALSE;
       "Logick_DB".PS_Sub := TRUE;
       #"Step" := #"Step" + 11;
   END_IF;
   #_w1 := (#"Step" = 21) AND NOT #Select_CMD;
   IF #_w1 THEN "PS_Main_DB".PS_One[#Select_PS].Mode := 5; END_IF;
   #_w2 := #_w1 AND ("PS_Main_DB".PS_One[#Select_PS].Mode = "PS_Main_DB".PS_One[#Select_PS].Status);
   IF #_w2 AND NOT "Logick_DB".Deload THEN
       #cnt := #cnt - 1;
       #"Step" := #"Step" + 1;
   END_IF;
   IF #_w2 AND "Logick_DB".Deload THEN #"Step" := #"Step" + 1; END_IF;
   #_w3 := #"Step" = 22;
   IF #_w3 THEN "PS_Main_DB".PS_One[#Select_PS].Mode := 6; END_IF;
   #_w4 := #_w3 AND ("PS_Main_DB".PS_One[#Select_PS].Mode = "PS_Main_DB".PS_One[#Select_PS].Status);
   IF #_w4 THEN
       "PS_Main_DB".PS_One[#Select_PS].CMD.Start_A := FALSE;
       #"Step" := #"Step" + 1;
   END_IF;
   #_w5 := (#"Step" >= 23) AND (#"Step" < 30);
   IF #_w5 THEN
       "Logick_DB".Deload := FALSE;
       "Logick_DB".PS_Sub := FALSE;
   END_IF;
   #T_Delay_OFF.Start := #_w5;
   IF #_w5 AND #T_Delay_OFF."Exit" THEN #"Step" := 10; END_IF;
   #T_Delay_OFF();   // "Time_M"
END_REGION

REGION Network 7: Ротация насосов
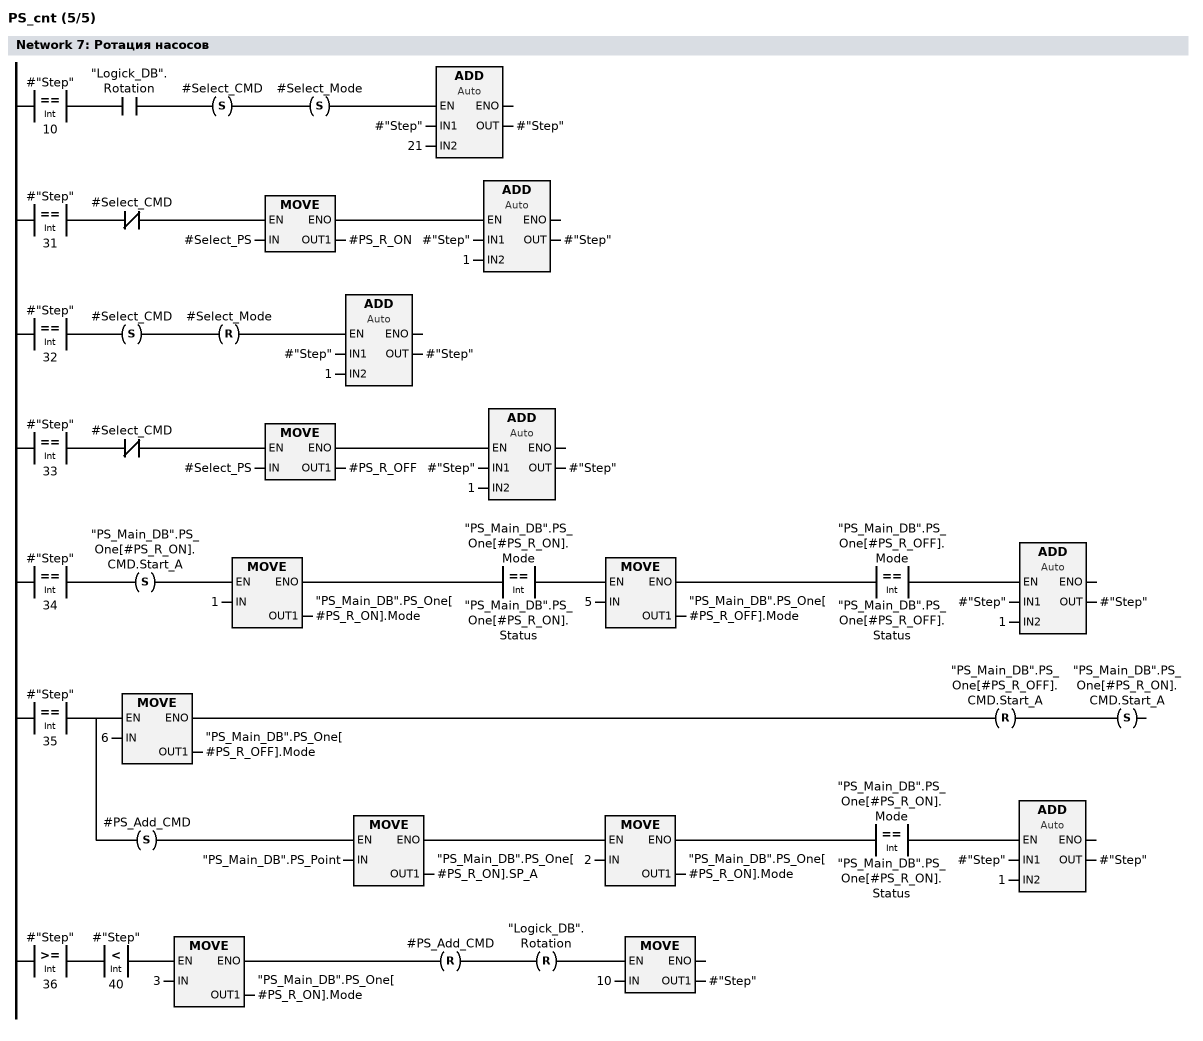
   RUNG wire#powerrail
      { S7_Templates := "SrcType := Int" } EQ_Contact(in1 := #"Step", in2 := 10)
      Contact( "Logick_DB".Rotation )
      S_Coil( #Select_CMD )
      S_Coil( #Select_Mode )
      Add(in1 := #"Step", in2 := 21, out => #"Step")
   END_RUNG
   RUNG wire#powerrail
      { S7_Templates := "SrcType := Int" } EQ_Contact(in1 := #"Step", in2 := 31)
      I_Contact( #Select_CMD )
      Move(in := #Select_PS, out1 => #PS_R_ON)
      Add(in1 := #"Step", in2 := 1, out => #"Step")
   END_RUNG
   RUNG wire#powerrail
      { S7_Templates := "SrcType := Int" } EQ_Contact(in1 := #"Step", in2 := 32)
      S_Coil( #Select_CMD )
      R_Coil( #Select_Mode )
      Add(in1 := #"Step", in2 := 1, out => #"Step")
   END_RUNG
   RUNG wire#powerrail
      { S7_Templates := "SrcType := Int" } EQ_Contact(in1 := #"Step", in2 := 33)
      I_Contact( #Select_CMD )
      Move(in := #Select_PS, out1 => #PS_R_OFF)
      Add(in1 := #"Step", in2 := 1, out => #"Step")
   END_RUNG
   RUNG wire#powerrail
      { S7_Templates := "SrcType := Int" } EQ_Contact(in1 := #"Step", in2 := 34)
      S_Coil( "PS_Main_DB".PS_One[#PS_R_ON].CMD.Start_A )
      Move(in := 1, out1 => "PS_Main_DB".PS_One[#PS_R_ON].Mode)
      { S7_Templates := "SrcType := Int" } EQ_Contact(in1 := "PS_Main_DB".PS_One[#PS_R_ON].Mode, in2 := "PS_Main_DB".PS_One[#PS_R_ON].Status)
      Move(in := 5, out1 => "PS_Main_DB".PS_One[#PS_R_OFF].Mode)
      { S7_Templates := "SrcType := Int" } EQ_Contact(in1 := "PS_Main_DB".PS_One[#PS_R_OFF].Mode, in2 := "PS_Main_DB".PS_One[#PS_R_OFF].Status)
      Add(in1 := #"Step", in2 := 1, out => #"Step")
   END_RUNG
   RUNG wire#powerrail
      { S7_Templates := "SrcType := Int" } EQ_Contact(in1 := #"Step", in2 := 35)
      wire#w1
      Move(in := 6, out1 => "PS_Main_DB".PS_One[#PS_R_OFF].Mode)
      R_Coil( "PS_Main_DB".PS_One[#PS_R_OFF].CMD.Start_A )
      S_Coil( "PS_Main_DB".PS_One[#PS_R_ON].CMD.Start_A )
   END_RUNG
   RUNG wire#w1
      S_Coil( #PS_Add_CMD )
      Move(in := "PS_Main_DB".PS_Point, out1 => "PS_Main_DB".PS_One[#PS_R_ON].SP_A)
      Move(in := 2, out1 => "PS_Main_DB".PS_One[#PS_R_ON].Mode)
      { S7_Templates := "SrcType := Int" } EQ_Contact(in1 := "PS_Main_DB".PS_One[#PS_R_ON].Mode, in2 := "PS_Main_DB".PS_One[#PS_R_ON].Status)
      Add(in1 := #"Step", in2 := 1, out => #"Step")
   END_RUNG
   RUNG wire#powerrail
      { S7_Templates := "SrcType := Int" } GE_Contact(in1 := #"Step", in2 := 36)
      { S7_Templates := "SrcType := Int" } LT_Contact(in1 := #"Step", in2 := 40)
      Move(in := 3, out1 => "PS_Main_DB".PS_One[#PS_R_ON].Mode)
      R_Coil( #PS_Add_CMD )
      R_Coil( "Logick_DB".Rotation )
      Move(in := 10, out1 => #"Step")
   END_RUNG
   // the same network as SCL:
   IF (#"Step" = 10) AND "Logick_DB".Rotation THEN
       #Select_CMD := TRUE;
       #Select_Mode := TRUE;
       #"Step" := #"Step" + 21;
   END_IF;
   IF (#"Step" = 31) AND NOT #Select_CMD THEN
       #PS_R_ON := #Select_PS;
       #"Step" := #"Step" + 1;
   END_IF;
   IF #"Step" = 32 THEN
       #Select_CMD := TRUE;
       #Select_Mode := FALSE;
       #"Step" := #"Step" + 1;
   END_IF;
   IF (#"Step" = 33) AND NOT #Select_CMD THEN
       #PS_R_OFF := #Select_PS;
       #"Step" := #"Step" + 1;
   END_IF;
   #_w1 := #"Step" = 34;
   IF #_w1 THEN
       "PS_Main_DB".PS_One[#PS_R_ON].CMD.Start_A := TRUE;
       "PS_Main_DB".PS_One[#PS_R_ON].Mode := 1;
   END_IF;
   #_w2 := #_w1 AND ("PS_Main_DB".PS_One[#PS_R_ON].Mode = "PS_Main_DB".PS_One[#PS_R_ON].Status);
   IF #_w2 THEN "PS_Main_DB".PS_One[#PS_R_OFF].Mode := 5; END_IF;
   IF #_w2 AND ("PS_Main_DB".PS_One[#PS_R_OFF].Mode = "PS_Main_DB".PS_One[#PS_R_OFF].Status) THEN
       #"Step" := #"Step" + 1;
   END_IF;
   #_w3 := #"Step" = 35;
   IF #_w3 THEN
       "PS_Main_DB".PS_One[#PS_R_OFF].Mode := 6;
       "PS_Main_DB".PS_One[#PS_R_OFF].CMD.Start_A := FALSE;
       "PS_Main_DB".PS_One[#PS_R_ON].CMD.Start_A := TRUE;
       #PS_Add_CMD := TRUE;
       "PS_Main_DB".PS_One[#PS_R_ON].SP_A := "PS_Main_DB".PS_Point;
       "PS_Main_DB".PS_One[#PS_R_ON].Mode := 2;
   END_IF;
   IF #_w3 AND ("PS_Main_DB".PS_One[#PS_R_ON].Mode = "PS_Main_DB".PS_One[#PS_R_ON].Status) THEN
       #"Step" := #"Step" + 1;
   END_IF;
   IF (#"Step" >= 36) AND (#"Step" < 40) THEN
       "PS_Main_DB".PS_One[#PS_R_ON].Mode := 3;
       #PS_Add_CMD := FALSE;
       "Logick_DB".Rotation := FALSE;
       #"Step" := 10;
   END_IF;
END_REGION
END_FUNCTION_BLOCK

FUNCTION "PS_Select" : Void
{ S7_Optimized_Access := 'TRUE' }
VERSION : 0.1
   VAR_INPUT 
      PS_All : Int;
   END_VAR

   VAR_IN_OUT 
      Weight : Real;
      CMD : Bool;
      Mode : Bool;   // 0 - останов, 1 - запуск
      PS_Number : Int;
   END_VAR

   VAR_TEMP 
      x : Int;
   END_VAR


BEGIN
	//контроль запроса на выбор насоса для запуска
	IF #CMD THEN
	    #Weight := 0.0;
	    #PS_Number := 0;
	    
	    FOR #x := 1 TO #PS_All DO
	        
	        //выбор максимального веса
	        IF "PS_Main_DB".PS_One[#x].Weight >= #Weight THEN
	            #Weight := "PS_Main_DB".PS_One[#x].Weight;
	        END_IF;
	        
	    END_FOR;
	    
	    //проходим по всему списку насосов
	    FOR #x := 1 TO #PS_All DO
	        
	        //выбор насоса для запуска
	        IF #Mode THEN
	            //проверяем приоритетность запуска для остановленных насосов
	            IF "PS_Main_DB".PS_One[#x].Weight <= #Weight AND "PS_Main_DB".PS_One[#x].CMD.Ready AND NOT "PS_Main_DB".PS_One[#x].CMD.Start_M THEN
	                #Weight := "PS_Main_DB".PS_One[#x].Weight;  //сохраняем приоритет в буфер
	                #PS_Number := #x;                           //возвращаем номер насоса для запуска
	            END_IF;
	        END_IF;
	        
	    END_FOR;
	    
	    FOR #x := 1 TO #PS_All DO
	        
	        //выбор максимального веса
	        IF "PS_Main_DB".PS_One[#x].Weight <= #Weight THEN
	            #Weight := "PS_Main_DB".PS_One[#x].Weight;
	        END_IF;
	        
	    END_FOR;
	    
	    //проходим по всему списку насосов
	    FOR #x := 1 TO #PS_All DO
	        
	        //выбор насоса для останова
	        IF NOT #Mode THEN
	            //проверяем приоритетность запуска для остановки насосов
	            IF "PS_Main_DB".PS_One[#x].Weight >= #Weight AND "PS_Main_DB".PS_One[#x].Status = 3 AND "PS_Main_DB".PS_One[#x].CMD.Start_M THEN
	                #Weight := "PS_Main_DB".PS_One[#x].Weight;  //сохраняем приоритет в буфер
	                #PS_Number := #x;                           //возвращаем номер насоса для запуска
	            END_IF;
	        END_IF;
	    END_FOR;
	    
	    //снятие флага запуска
	    #CMD := FALSE;
	END_IF;
	
	
	
	
	
END_FUNCTION

FUNCTION_BLOCK "PS_One"   // FB11, LAD
{ S7_Optimized_Access := 'FALSE' }
VERSION : 0.1
// Mode - 0 - выкл, 1 - быстрый разгон, 2 - плавный разон, 3 - работа, 4 - притормозить для ввода нового насоса, 5 - замедлить плавно, 6 - замедлить быстро
// 
// Status - 0 выкл, 1 - быстро разгоняется, 10 - вышел на точку, 2 - плавно разгоняется, 20 - вышел на точку, 3 - в работе, 4 - притормаживается для выхода на общую точку, 40 - общая точка достигнута, 5 - замедлить для отключения, 50 - замедлено до нижней точки, 6 - вывести из работы через быстрый сброс оборотов, 60 - обороты сброшены и готов к отключению, 99 - насос в аварии/не готов к работе
// stored: AutoNumber false, IsIECCheckEnabled false, SetENOAutomatically false, UDAEnableTagReadback false
   VAR_INPUT
      in_PE : Real;   // Давление на всасывании
      P_FB_SP : Real;   // Текущая скорость / Уставка скорости для ЧП
      P_Alarm : Bool;   // Авария ЧП
      P_Warning : Bool;   // Предупреждение ЧП
   END_VAR
   VAR_OUTPUT
      P_CMD : Bool;   // Команда на ЧП
      P_SP : Real;   // Уставка на ЧП
      P_Step_Up : Real := 0.01;   // Шаг разгона для ЧП
      P_Step_Down : Real := 0.01;   // Шаг замедления для ЧП
   END_VAR
   VAR_IN_OUT
      P_Res : DInt;   // Наработка ЧП
   END_VAR
   VAR DB_SPECIFIC
      CMD : "CMD";   // Блок команд
      Min { S7_SetPoint := 'True'} : Bool;
      Max : Bool;
      PE_Warning : Bool;
      SP_A : Real;   // Уставка в авторежиме
      SP : Real;   // Фактическая уставка
      Mode : Int;   // Запрашиваемый режим работы
      Hand_Mode : Int := 3;   // Режим работы в ручном режиме
      Status : Int;   // Фактический режим работы
      Weight : Real;   // Коэфф. выбора насоса
      Start_per_H_SP : Int := 5;
      Start_per_H_Now : Int;
      Alarms : Word;
      Events : Word;
      pos : Array[0..15] of Bool;
   END_VAR
   VAR
      T_Delay { S7_SetPoint := 'True'} : "Time_M";   // Минимальная задержка между пусками
      T_PE_Delay { S7_SetPoint := 'True'} : "Time_M";
   END_VAR
   VAR_TEMP
      ev : Bool;
   END_VAR
   // T_Delay.SP_M := 10;
   // T_Delay.SP_S := 0;
   VAR_TEMP   // added for the SCL form of the ladder/FBD networks
      _w1 : Bool;
      _w2 : Bool;
      _w3 : Bool;
      _w4 : Bool;
      _w5 : Bool;
      _w6 : Bool;
      _w7 : Bool;
      _w8 : Bool;
      _w9 : Bool;
      _w10 : Bool;
      _w11 : Bool;
      _w12 : Bool;
      _w13 : Bool;
      _w14 : Bool;
      _w15 : Bool;
      _w16 : Bool;
      _w17 : Bool;
      _w18 : Bool;
      _w19 : Bool;
      _w20 : Bool;
   END_VAR
BEGIN

REGION Network 1: - - -
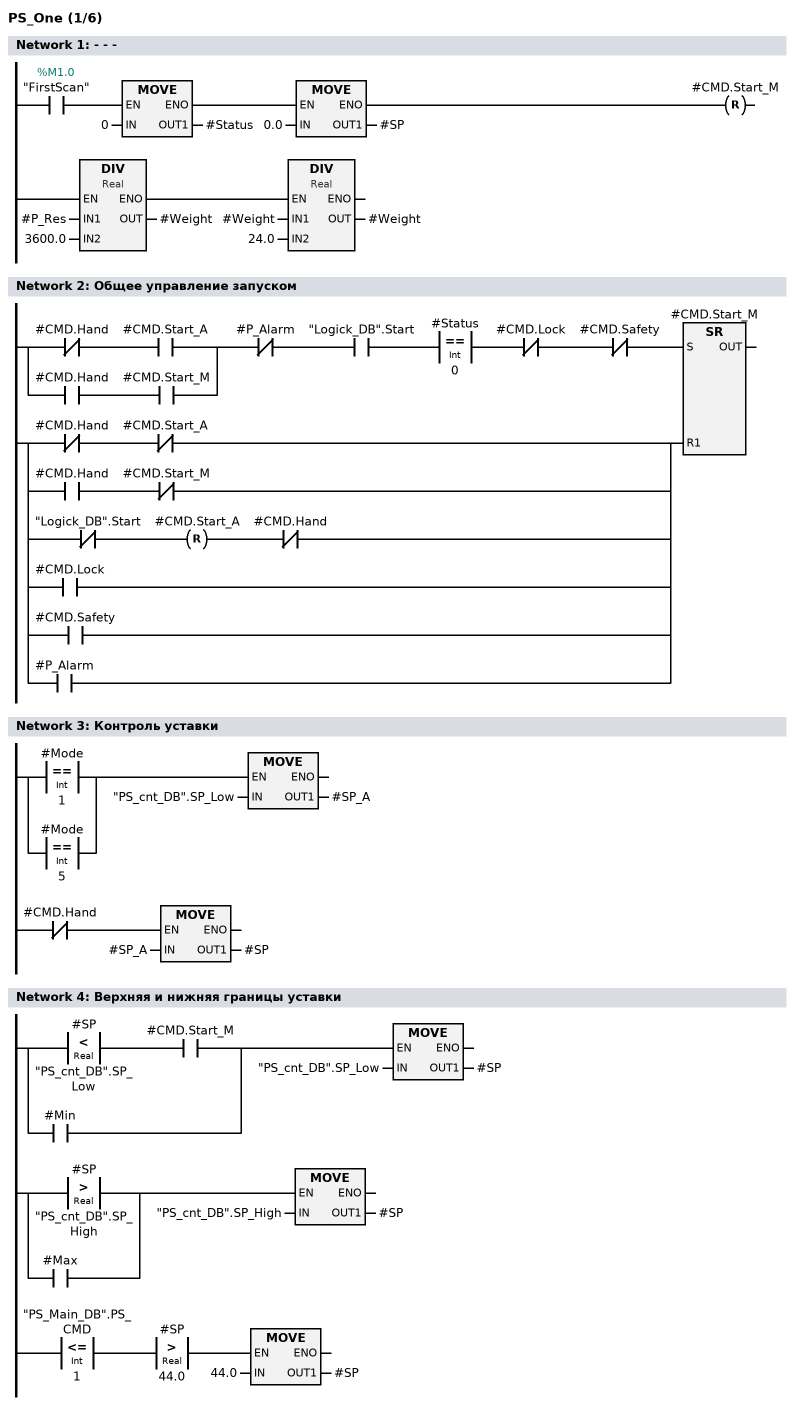
   RUNG wire#powerrail
      Contact( "FirstScan" )
      Move(in := 0, out1 => #Status)
      Move(in := 0.0, out1 => #SP)
      R_Coil( #CMD.Start_M )
   END_RUNG
   RUNG wire#powerrail
      { S7_Templates := "SrcType := Real" } Div(in1 := #P_Res, in2 := 3600.0, out => #Weight)
      { S7_Templates := "SrcType := Real" } Div(in1 := #Weight, in2 := 24.0, out => #Weight)
   END_RUNG
   // the same network as SCL:
   IF "FirstScan" THEN
       #Status := 0;
       #SP := 0.0;
       #CMD.Start_M := FALSE;
   END_IF;
   #Weight := #P_Res / 3600.0;
   #Weight := #Weight / 24.0;
END_REGION

REGION Network 2: Общее управление запуском
   RUNG wire#powerrail
      I_Contact( #CMD.Hand )
      Contact( #CMD.Start_A )
      wire#w1
      I_Contact( #P_Alarm )
      Contact( "Logick_DB".Start )
      { S7_Templates := "SrcType := Int" } EQ_Contact(in1 := #Status, in2 := 0)
      I_Contact( #CMD.Lock )
      I_Contact( #CMD.Safety )
      S_SR(operand := #CMD.Start_M, r1 := wire#w2)
   END_RUNG
   RUNG wire#powerrail
      Contact( #CMD.Hand )
      Contact( #CMD.Start_M )
   END_RUNG wire#w1
   RUNG wire#powerrail
      I_Contact( #CMD.Hand )
      I_Contact( #CMD.Start_A )
   END_RUNG wire#w2
   RUNG wire#powerrail
      Contact( #CMD.Hand )
      I_Contact( #CMD.Start_M )
   END_RUNG wire#w2
   RUNG wire#powerrail
      I_Contact( "Logick_DB".Start )
      R_Coil( #CMD.Start_A )
      I_Contact( #CMD.Hand )
   END_RUNG wire#w2
   RUNG wire#powerrail
      Contact( #CMD.Lock )
   END_RUNG wire#w2
   RUNG wire#powerrail
      Contact( #CMD.Safety )
   END_RUNG wire#w2
   RUNG wire#powerrail
      Contact( #P_Alarm )
   END_RUNG wire#w2
   // the same network as SCL:
   #_w1 := ((NOT #CMD.Hand AND #CMD.Start_A) OR (#CMD.Hand AND #CMD.Start_M)) AND NOT #P_Alarm AND "Logick_DB".Start AND (#Status = 0) AND NOT #CMD.Lock AND NOT #CMD.Safety;
   #_w2 := NOT #CMD.Hand AND NOT #CMD.Start_A;
   IF NOT "Logick_DB".Start THEN #CMD.Start_A := FALSE; END_IF;
   #_w3 := #_w2 OR (#CMD.Hand AND NOT #CMD.Start_M) OR (NOT "Logick_DB".Start AND NOT #CMD.Hand) OR #CMD.Lock OR #CMD.Safety OR #P_Alarm;
   IF #_w1 THEN
       #CMD.Start_M := TRUE;   // SR flip-flop
   END_IF;
   IF #_w3 THEN #CMD.Start_M := FALSE; END_IF;
END_REGION

REGION Network 3: Контроль уставки
   RUNG wire#powerrail
      { S7_Templates := "SrcType := Int" } EQ_Contact(in1 := #Mode, in2 := 1)
      wire#w1
      Move(in := "PS_cnt_DB".SP_Low, out1 => #SP_A)
   END_RUNG
   RUNG wire#powerrail
      { S7_Templates := "SrcType := Int" } EQ_Contact(in1 := #Mode, in2 := 5)
   END_RUNG wire#w1
   RUNG wire#powerrail
      I_Contact( #CMD.Hand )
      Move(in := #SP_A, out1 => #SP)
   END_RUNG
   // the same network as SCL:
   IF (#Mode = 1) OR (#Mode = 5) THEN #SP_A := "PS_cnt_DB".SP_Low; END_IF;
   IF NOT #CMD.Hand THEN #SP := #SP_A; END_IF;
END_REGION

REGION Network 4: Верхняя и нижняя границы уставки
   RUNG wire#powerrail
      { S7_Templates := "SrcType := Real" } LT_Contact(in1 := #SP, in2 := "PS_cnt_DB".SP_Low)
      Contact( #CMD.Start_M )
      wire#w1
      Move(in := "PS_cnt_DB".SP_Low, out1 => #SP)
   END_RUNG
   RUNG wire#powerrail
      Contact( #Min )
   END_RUNG wire#w1
   RUNG wire#powerrail
      { S7_Templates := "SrcType := Real" } GT_Contact(in1 := #SP, in2 := "PS_cnt_DB".SP_High)
      wire#w2
      Move(in := "PS_cnt_DB".SP_High, out1 => #SP)
   END_RUNG
   RUNG wire#powerrail
      Contact( #Max )
   END_RUNG wire#w2
   RUNG wire#powerrail
      { S7_Templates := "SrcType := Int" } LE_Contact(in1 := "PS_Main_DB".PS_CMD, in2 := 1)
      { S7_Templates := "SrcType := Real" } GT_Contact(in1 := #SP, in2 := 44.0)
      Move(in := 44.0, out1 => #SP)
   END_RUNG
   // the same network as SCL:
   IF ((#SP < "PS_cnt_DB".SP_Low) AND #CMD.Start_M) OR #Min THEN #SP := "PS_cnt_DB".SP_Low; END_IF;
   IF (#SP > "PS_cnt_DB".SP_High) OR #Max THEN #SP := "PS_cnt_DB".SP_High; END_IF;
   IF ("PS_Main_DB".PS_CMD <= 1) AND (#SP > 44.0) THEN #SP := 44.0; END_IF;
END_REGION

REGION Network 5
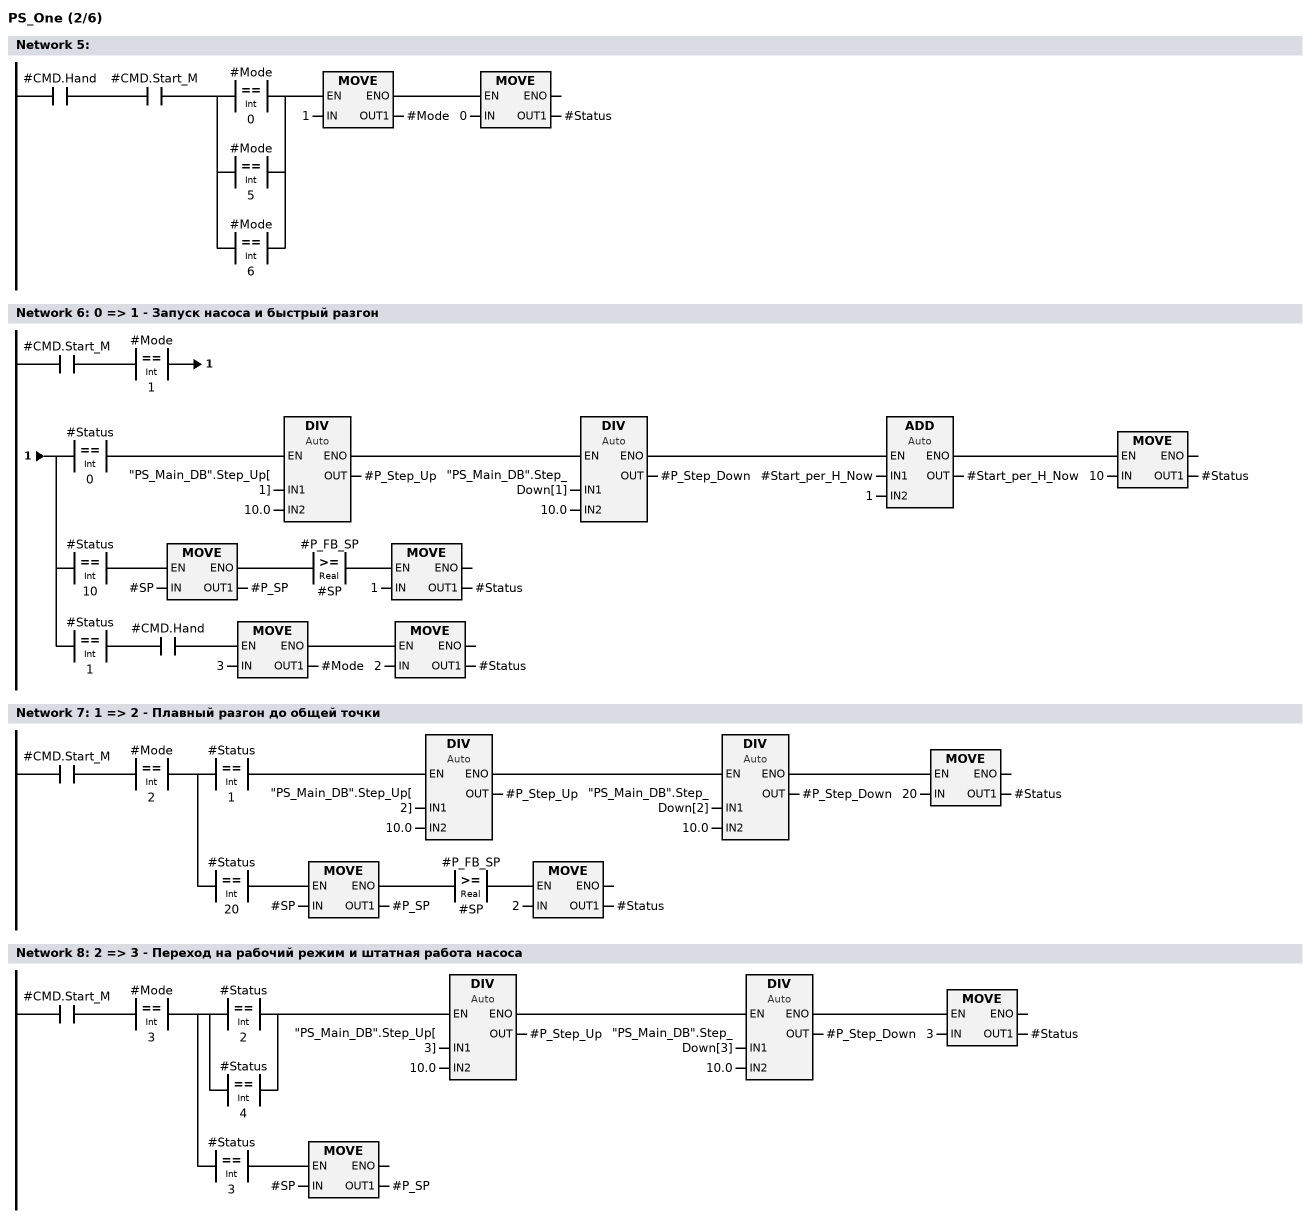
   RUNG wire#powerrail
      Contact( #CMD.Hand )
      Contact( #CMD.Start_M )
      wire#w1
      { S7_Templates := "SrcType := Int" } EQ_Contact(in1 := #Mode, in2 := 0)
      wire#w2
      Move(in := 1, out1 => #Mode)
      Move(in := 0, out1 => #Status)
   END_RUNG
   RUNG wire#w1
      { S7_Templates := "SrcType := Int" } EQ_Contact(in1 := #Mode, in2 := 5)
   END_RUNG wire#w2
   RUNG wire#w1
      { S7_Templates := "SrcType := Int" } EQ_Contact(in1 := #Mode, in2 := 6)
   END_RUNG wire#w2
   // the same network as SCL:
   #_w1 := #CMD.Hand AND #CMD.Start_M AND ((#Mode = 0) OR (#Mode = 5) OR (#Mode = 6));
   IF #_w1 THEN
       #Mode := 1;
       #Status := 0;
   END_IF;
END_REGION

REGION Network 6: 0 => 1 - Запуск насоса и быстрый разгон
   RUNG wire#powerrail
      Contact( #CMD.Start_M )
      { S7_Templates := "SrcType := Int" } EQ_Contact(in1 := #Mode, in2 := 1)
      wire#w1
      { S7_Templates := "SrcType := Int" } EQ_Contact(in1 := #Status, in2 := 0)
      Div(in1 := "PS_Main_DB".Step_Up[1], in2 := 10.0, out => #P_Step_Up)
      Div(in1 := "PS_Main_DB".Step_Down[1], in2 := 10.0, out => #P_Step_Down)
      Add(in1 := #Start_per_H_Now, in2 := 1, out => #Start_per_H_Now)
      Move(in := 10, out1 => #Status)
   END_RUNG
   RUNG wire#w1
      { S7_Templates := "SrcType := Int" } EQ_Contact(in1 := #Status, in2 := 10)
      Move(in := #SP, out1 => #P_SP)
      { S7_Templates := "SrcType := Real" } GE_Contact(in1 := #P_FB_SP, in2 := #SP)
      Move(in := 1, out1 => #Status)
   END_RUNG
   RUNG wire#w1
      { S7_Templates := "SrcType := Int" } EQ_Contact(in1 := #Status, in2 := 1)
      Contact( #CMD.Hand )
      Move(in := 3, out1 => #Mode)
      Move(in := 2, out1 => #Status)
   END_RUNG
   // the same network as SCL:
   #_w1 := #CMD.Start_M AND (#Mode = 1);
   IF #_w1 AND (#Status = 0) THEN
       #P_Step_Up := "PS_Main_DB".Step_Up[1] / 10.0;
       #P_Step_Down := "PS_Main_DB".Step_Down[1] / 10.0;
       #Start_per_H_Now := #Start_per_H_Now + 1;
       #Status := 10;
   END_IF;
   #_w2 := #_w1 AND (#Status = 10);
   IF #_w2 THEN #P_SP := #SP; END_IF;
   IF #_w2 AND (#P_FB_SP >= #SP) THEN #Status := 1; END_IF;
   IF #_w1 AND (#Status = 1) AND #CMD.Hand THEN
       #Mode := 3;
       #Status := 2;
   END_IF;
END_REGION

REGION Network 7: 1 => 2 - Плавный разгон до общей точки
   RUNG wire#powerrail
      Contact( #CMD.Start_M )
      { S7_Templates := "SrcType := Int" } EQ_Contact(in1 := #Mode, in2 := 2)
      wire#w1
      { S7_Templates := "SrcType := Int" } EQ_Contact(in1 := #Status, in2 := 1)
      Div(in1 := "PS_Main_DB".Step_Up[2], in2 := 10.0, out => #P_Step_Up)
      Div(in1 := "PS_Main_DB".Step_Down[2], in2 := 10.0, out => #P_Step_Down)
      Move(in := 20, out1 => #Status)
   END_RUNG
   RUNG wire#w1
      { S7_Templates := "SrcType := Int" } EQ_Contact(in1 := #Status, in2 := 20)
      Move(in := #SP, out1 => #P_SP)
      { S7_Templates := "SrcType := Real" } GE_Contact(in1 := #P_FB_SP, in2 := #SP)
      Move(in := 2, out1 => #Status)
   END_RUNG
   // the same network as SCL:
   #_w1 := #CMD.Start_M AND (#Mode = 2);
   IF #_w1 AND (#Status = 1) THEN
       #P_Step_Up := "PS_Main_DB".Step_Up[2] / 10.0;
       #P_Step_Down := "PS_Main_DB".Step_Down[2] / 10.0;
       #Status := 20;
   END_IF;
   #_w2 := #_w1 AND (#Status = 20);
   IF #_w2 THEN #P_SP := #SP; END_IF;
   IF #_w2 AND (#P_FB_SP >= #SP) THEN #Status := 2; END_IF;
END_REGION

REGION Network 8: 2 => 3 - Переход на рабочий режим и штатная работа насоса
   RUNG wire#powerrail
      Contact( #CMD.Start_M )
      { S7_Templates := "SrcType := Int" } EQ_Contact(in1 := #Mode, in2 := 3)
      wire#w1
      { S7_Templates := "SrcType := Int" } EQ_Contact(in1 := #Status, in2 := 2)
      wire#w2
      Div(in1 := "PS_Main_DB".Step_Up[3], in2 := 10.0, out => #P_Step_Up)
      Div(in1 := "PS_Main_DB".Step_Down[3], in2 := 10.0, out => #P_Step_Down)
      Move(in := 3, out1 => #Status)
   END_RUNG
   RUNG wire#w1
      { S7_Templates := "SrcType := Int" } EQ_Contact(in1 := #Status, in2 := 4)
   END_RUNG wire#w2
   RUNG wire#w1
      { S7_Templates := "SrcType := Int" } EQ_Contact(in1 := #Status, in2 := 3)
      Move(in := #SP, out1 => #P_SP)
   END_RUNG
   // the same network as SCL:
   #_w1 := #CMD.Start_M AND (#Mode = 3);
   IF #_w1 AND ((#Status = 2) OR (#Status = 4)) THEN
       #P_Step_Up := "PS_Main_DB".Step_Up[3] / 10.0;
       #P_Step_Down := "PS_Main_DB".Step_Down[3] / 10.0;
       #Status := 3;
   END_IF;
   IF #_w1 AND (#Status = 3) THEN #P_SP := #SP; END_IF;
END_REGION

REGION Network 9: 3 => 4 - Снижение скорости для подключения нового насоса
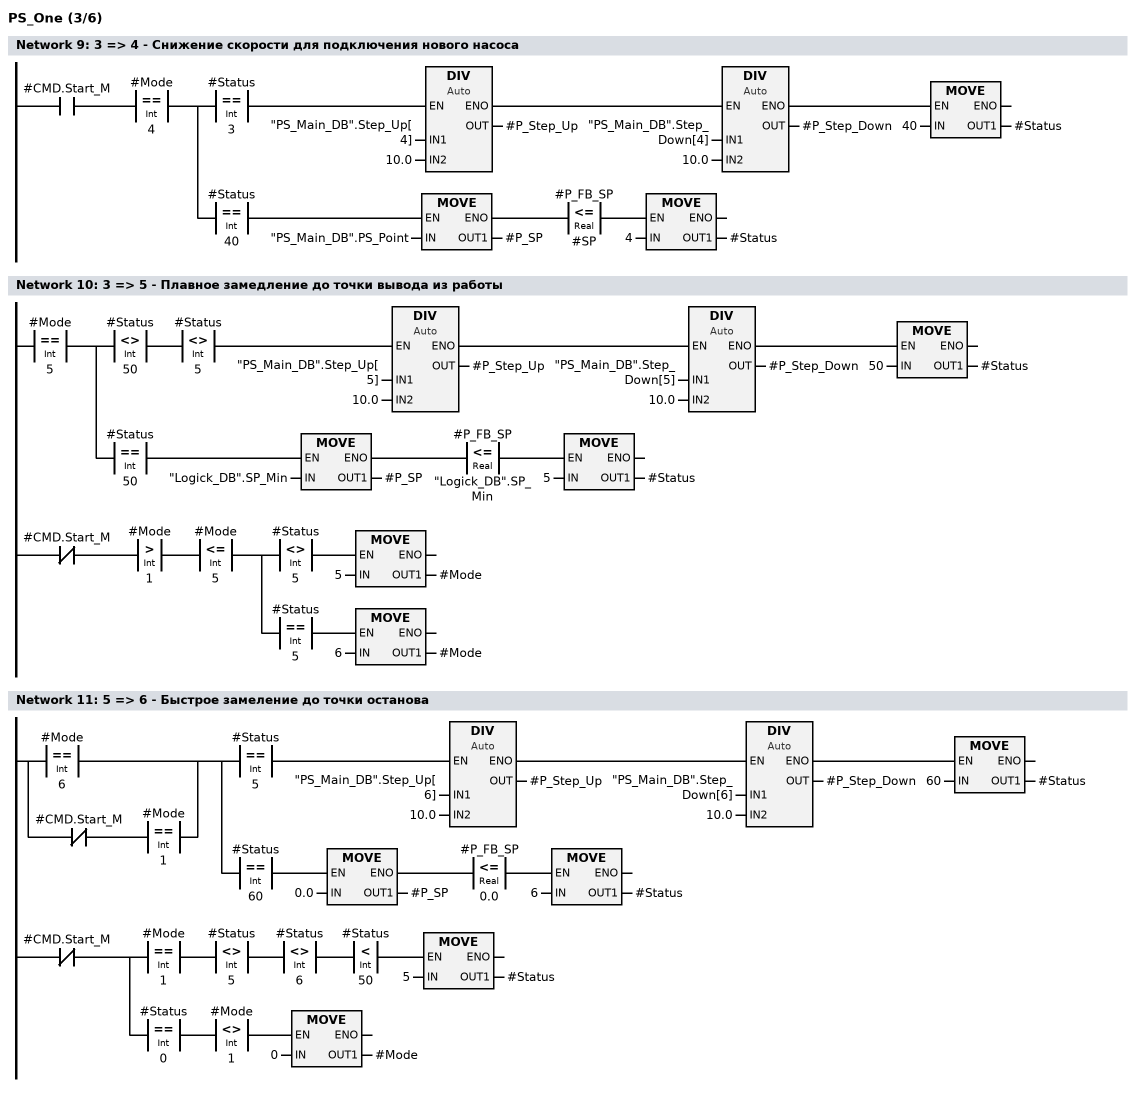
   RUNG wire#powerrail
      Contact( #CMD.Start_M )
      { S7_Templates := "SrcType := Int" } EQ_Contact(in1 := #Mode, in2 := 4)
      wire#w1
      { S7_Templates := "SrcType := Int" } EQ_Contact(in1 := #Status, in2 := 3)
      Div(in1 := "PS_Main_DB".Step_Up[4], in2 := 10.0, out => #P_Step_Up)
      Div(in1 := "PS_Main_DB".Step_Down[4], in2 := 10.0, out => #P_Step_Down)
      Move(in := 40, out1 => #Status)
   END_RUNG
   RUNG wire#w1
      { S7_Templates := "SrcType := Int" } EQ_Contact(in1 := #Status, in2 := 40)
      Move(in := "PS_Main_DB".PS_Point, out1 => #P_SP)
      { S7_Templates := "SrcType := Real" } LE_Contact(in1 := #P_FB_SP, in2 := #SP)
      Move(in := 4, out1 => #Status)
   END_RUNG
   // the same network as SCL:
   #_w1 := #CMD.Start_M AND (#Mode = 4);
   IF #_w1 AND (#Status = 3) THEN
       #P_Step_Up := "PS_Main_DB".Step_Up[4] / 10.0;
       #P_Step_Down := "PS_Main_DB".Step_Down[4] / 10.0;
       #Status := 40;
   END_IF;
   #_w2 := #_w1 AND (#Status = 40);
   IF #_w2 THEN #P_SP := "PS_Main_DB".PS_Point; END_IF;
   IF #_w2 AND (#P_FB_SP <= #SP) THEN #Status := 4; END_IF;
END_REGION

REGION Network 10: 3 => 5 - Плавное замедление до точки вывода из работы
   RUNG wire#powerrail
      { S7_Templates := "SrcType := Int" } EQ_Contact(in1 := #Mode, in2 := 5)
      wire#w1
      { S7_Templates := "SrcType := Int" } NE_Contact(in1 := #Status, in2 := 50)
      { S7_Templates := "SrcType := Int" } NE_Contact(in1 := #Status, in2 := 5)
      Div(in1 := "PS_Main_DB".Step_Up[5], in2 := 10.0, out => #P_Step_Up)
      Div(in1 := "PS_Main_DB".Step_Down[5], in2 := 10.0, out => #P_Step_Down)
      Move(in := 50, out1 => #Status)
   END_RUNG
   RUNG wire#w1
      { S7_Templates := "SrcType := Int" } EQ_Contact(in1 := #Status, in2 := 50)
      Move(in := "Logick_DB".SP_Min, out1 => #P_SP)
      { S7_Templates := "SrcType := Real" } LE_Contact(in1 := #P_FB_SP, in2 := "Logick_DB".SP_Min)
      Move(in := 5, out1 => #Status)
   END_RUNG
   RUNG wire#powerrail
      I_Contact( #CMD.Start_M )
      { S7_Templates := "SrcType := Int" } GT_Contact(in1 := #Mode, in2 := 1)
      { S7_Templates := "SrcType := Int" } LE_Contact(in1 := #Mode, in2 := 5)
      wire#w2
      { S7_Templates := "SrcType := Int" } NE_Contact(in1 := #Status, in2 := 5)
      Move(in := 5, out1 => #Mode)
   END_RUNG
   RUNG wire#w2
      { S7_Templates := "SrcType := Int" } EQ_Contact(in1 := #Status, in2 := 5)
      Move(in := 6, out1 => #Mode)
   END_RUNG
   // the same network as SCL:
   #_w1 := #Mode = 5;
   IF #_w1 AND (#Status <> 50) AND (#Status <> 5) THEN
       #P_Step_Up := "PS_Main_DB".Step_Up[5] / 10.0;
       #P_Step_Down := "PS_Main_DB".Step_Down[5] / 10.0;
       #Status := 50;
   END_IF;
   #_w2 := #_w1 AND (#Status = 50);
   IF #_w2 THEN #P_SP := "Logick_DB".SP_Min; END_IF;
   IF #_w2 AND (#P_FB_SP <= "Logick_DB".SP_Min) THEN #Status := 5; END_IF;
   #_w3 := NOT #CMD.Start_M AND (#Mode > 1) AND (#Mode <= 5);
   IF #_w3 AND (#Status <> 5) THEN #Mode := 5; END_IF;
   IF #_w3 AND (#Status = 5) THEN #Mode := 6; END_IF;
END_REGION

REGION Network 11: 5 => 6 - Быстрое замеление до точки останова
   RUNG wire#powerrail
      { S7_Templates := "SrcType := Int" } EQ_Contact(in1 := #Mode, in2 := 6)
      wire#w1
      { S7_Templates := "SrcType := Int" } EQ_Contact(in1 := #Status, in2 := 5)
      Div(in1 := "PS_Main_DB".Step_Up[6], in2 := 10.0, out => #P_Step_Up)
      Div(in1 := "PS_Main_DB".Step_Down[6], in2 := 10.0, out => #P_Step_Down)
      Move(in := 60, out1 => #Status)
   END_RUNG
   RUNG wire#powerrail
      I_Contact( #CMD.Start_M )
      { S7_Templates := "SrcType := Int" } EQ_Contact(in1 := #Mode, in2 := 1)
   END_RUNG wire#w1
   RUNG wire#w1
      { S7_Templates := "SrcType := Int" } EQ_Contact(in1 := #Status, in2 := 60)
      Move(in := 0.0, out1 => #P_SP)
      { S7_Templates := "SrcType := Real" } LE_Contact(in1 := #P_FB_SP, in2 := 0.0)
      Move(in := 6, out1 => #Status)
   END_RUNG
   RUNG wire#powerrail
      I_Contact( #CMD.Start_M )
      wire#w2
      { S7_Templates := "SrcType := Int" } EQ_Contact(in1 := #Mode, in2 := 1)
      { S7_Templates := "SrcType := Int" } NE_Contact(in1 := #Status, in2 := 5)
      { S7_Templates := "SrcType := Int" } NE_Contact(in1 := #Status, in2 := 6)
      { S7_Templates := "SrcType := Int" } LT_Contact(in1 := #Status, in2 := 50)
      Move(in := 5, out1 => #Status)
   END_RUNG
   RUNG wire#w2
      { S7_Templates := "SrcType := Int" } EQ_Contact(in1 := #Status, in2 := 0)
      { S7_Templates := "SrcType := Int" } NE_Contact(in1 := #Mode, in2 := 1)
      Move(in := 0, out1 => #Mode)
   END_RUNG
   // the same network as SCL:
   #_w1 := (#Mode = 6) OR (NOT #CMD.Start_M AND (#Mode = 1));
   IF #_w1 AND (#Status = 5) THEN
       #P_Step_Up := "PS_Main_DB".Step_Up[6] / 10.0;
       #P_Step_Down := "PS_Main_DB".Step_Down[6] / 10.0;
       #Status := 60;
   END_IF;
   #_w2 := #_w1 AND (#Status = 60);
   IF #_w2 THEN #P_SP := 0.0; END_IF;
   IF #_w2 AND (#P_FB_SP <= 0.0) THEN #Status := 6; END_IF;
   IF NOT #CMD.Start_M AND (#Mode = 1) AND (#Status <> 5) AND (#Status <> 6) AND (#Status < 50) THEN
       #Status := 5;
   END_IF;
   IF NOT #CMD.Start_M AND (#Status = 0) AND (#Mode <> 1) THEN #Mode := 0; END_IF;
END_REGION

REGION Network 12: 6 => 0 - Насос успешно остановлен
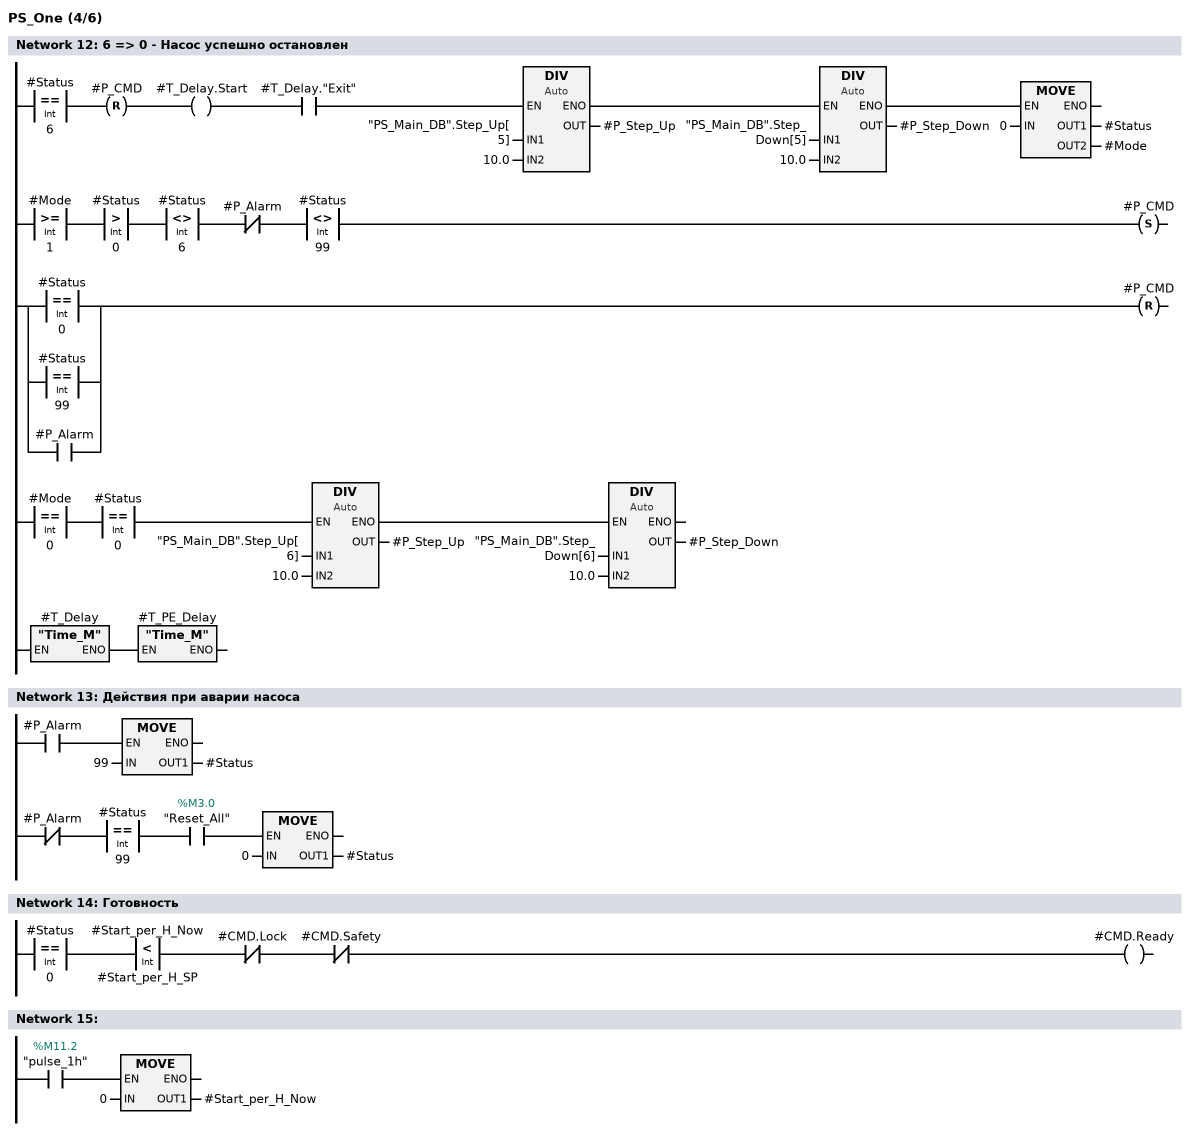
   RUNG wire#powerrail
      { S7_Templates := "SrcType := Int" } EQ_Contact(in1 := #Status, in2 := 6)
      R_Coil( #P_CMD )
      Coil( #T_Delay.Start )
      Contact( #T_Delay."Exit" )
      Div(in1 := "PS_Main_DB".Step_Up[5], in2 := 10.0, out => #P_Step_Up)
      Div(in1 := "PS_Main_DB".Step_Down[5], in2 := 10.0, out => #P_Step_Down)
      Move(in := 0, out1 => #Status, out2 => #Mode)
   END_RUNG
   RUNG wire#powerrail
      { S7_Templates := "SrcType := Int" } GE_Contact(in1 := #Mode, in2 := 1)
      { S7_Templates := "SrcType := Int" } GT_Contact(in1 := #Status, in2 := 0)
      { S7_Templates := "SrcType := Int" } NE_Contact(in1 := #Status, in2 := 6)
      I_Contact( #P_Alarm )
      { S7_Templates := "SrcType := Int" } NE_Contact(in1 := #Status, in2 := 99)
      S_Coil( #P_CMD )
   END_RUNG
   RUNG wire#powerrail
      { S7_Templates := "SrcType := Int" } EQ_Contact(in1 := #Status, in2 := 0)
      wire#w1
      R_Coil( #P_CMD )
   END_RUNG
   RUNG wire#powerrail
      { S7_Templates := "SrcType := Int" } EQ_Contact(in1 := #Status, in2 := 99)
   END_RUNG wire#w1
   RUNG wire#powerrail
      Contact( #P_Alarm )
   END_RUNG wire#w1
   RUNG wire#powerrail
      { S7_Templates := "SrcType := Int" } EQ_Contact(in1 := #Mode, in2 := 0)
      { S7_Templates := "SrcType := Int" } EQ_Contact(in1 := #Status, in2 := 0)
      Div(in1 := "PS_Main_DB".Step_Up[6], in2 := 10.0, out => #P_Step_Up)
      Div(in1 := "PS_Main_DB".Step_Down[6], in2 := 10.0, out => #P_Step_Down)
   END_RUNG
   RUNG wire#powerrail
      #T_Delay()
      #T_PE_Delay()
   END_RUNG
   // the same network as SCL:
   #_w1 := #Status = 6;
   IF #_w1 THEN #P_CMD := FALSE; END_IF;
   #T_Delay.Start := #_w1;
   IF #_w1 AND #T_Delay."Exit" THEN
       #P_Step_Up := "PS_Main_DB".Step_Up[5] / 10.0;
       #P_Step_Down := "PS_Main_DB".Step_Down[5] / 10.0;
       #Status := 0;
       #Mode := 0;
   END_IF;
   IF (#Mode >= 1) AND (#Status > 0) AND (#Status <> 6) AND NOT #P_Alarm AND (#Status <> 99) THEN
       #P_CMD := TRUE;
   END_IF;
   IF (#Status = 0) OR (#Status = 99) OR #P_Alarm THEN #P_CMD := FALSE; END_IF;
   IF (#Mode = 0) AND (#Status = 0) THEN
       #P_Step_Up := "PS_Main_DB".Step_Up[6] / 10.0;
       #P_Step_Down := "PS_Main_DB".Step_Down[6] / 10.0;
   END_IF;
   #T_Delay(ENO => #_w2);   // "Time_M"
   IF #_w2 THEN
       #T_PE_Delay();   // "Time_M"
   END_IF;
END_REGION

REGION Network 13: Действия при аварии насоса
   RUNG wire#powerrail
      Contact( #P_Alarm )
      Move(in := 99, out1 => #Status)
   END_RUNG
   RUNG wire#powerrail
      I_Contact( #P_Alarm )
      { S7_Templates := "SrcType := Int" } EQ_Contact(in1 := #Status, in2 := 99)
      Contact( "Reset_All" )
      Move(in := 0, out1 => #Status)
   END_RUNG
   // the same network as SCL:
   IF #P_Alarm THEN #Status := 99; END_IF;
   IF NOT #P_Alarm AND (#Status = 99) AND "Reset_All" THEN #Status := 0; END_IF;
END_REGION

REGION Network 14: Готовность
   RUNG wire#powerrail
      { S7_Templates := "SrcType := Int" } EQ_Contact(in1 := #Status, in2 := 0)
      { S7_Templates := "SrcType := Int" } LT_Contact(in1 := #Start_per_H_Now, in2 := #Start_per_H_SP)
      I_Contact( #CMD.Lock )
      I_Contact( #CMD.Safety )
      Coil( #CMD.Ready )
   END_RUNG
   // the same network as SCL:
   #CMD.Ready := (#Status = 0) AND (#Start_per_H_Now < #Start_per_H_SP) AND NOT #CMD.Lock AND NOT #CMD.Safety;
END_REGION

REGION Network 15
   RUNG wire#powerrail
      Contact( "pulse_1h" )
      Move(in := 0, out1 => #Start_per_H_Now)
   END_RUNG
   // the same network as SCL:
   IF "pulse_1h" THEN #Start_per_H_Now := 0; END_IF;
END_REGION

REGION Network 16
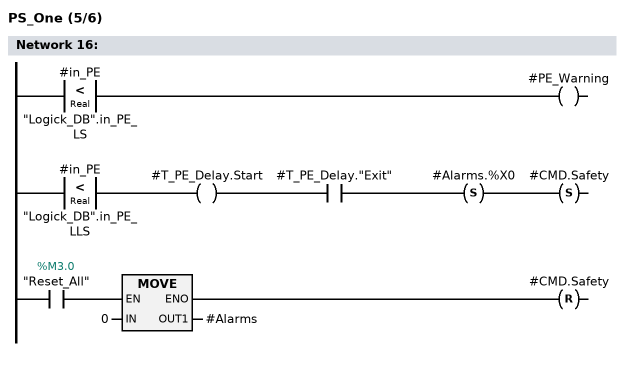
   RUNG wire#powerrail
      { S7_Templates := "SrcType := Real" } LT_Contact(in1 := #in_PE, in2 := "Logick_DB".in_PE_LS)
      Coil( #PE_Warning )
   END_RUNG
   RUNG wire#powerrail
      { S7_Templates := "SrcType := Real" } LT_Contact(in1 := #in_PE, in2 := "Logick_DB".in_PE_LLS)
      Coil( #T_PE_Delay.Start )
      Contact( #T_PE_Delay."Exit" )
      S_Coil( #Alarms.%X0 )
      S_Coil( #CMD.Safety )
   END_RUNG
   RUNG wire#powerrail
      Contact( "Reset_All" )
      Move(in := 0, out1 => #Alarms)
      R_Coil( #CMD.Safety )
   END_RUNG
   // the same network as SCL:
   #PE_Warning := #in_PE < "Logick_DB".in_PE_LS;
   #T_PE_Delay.Start := #in_PE < "Logick_DB".in_PE_LLS;
   IF #T_PE_Delay.Start AND #T_PE_Delay."Exit" THEN
       #Alarms.%X0 := TRUE;
       #CMD.Safety := TRUE;
   END_IF;
   IF "Reset_All" THEN
       #Alarms := 0;
       #CMD.Safety := FALSE;
   END_IF;
END_REGION

REGION Network 17: События привода
   // 0 - ручной режим активирован
   // 1 - ручной режим деактивирован
   // 2 - принудительный режим активирован
   // 3 - принудительный режим деактивирован
   // 4 - запуск в ручном режиме
   // 5 - останов в ручном режиме
   // 6 - местный режим управления активирован
   // 7 - местный режим управления деактивирован
   // 8 - запущено в местном режиме
   // 9 - остановлено в местном режиме
   // 10 - сервисный режим активирован
   // 11 - сервисный режим деактивирован
   // 12 - проведено сервисное обслуживание
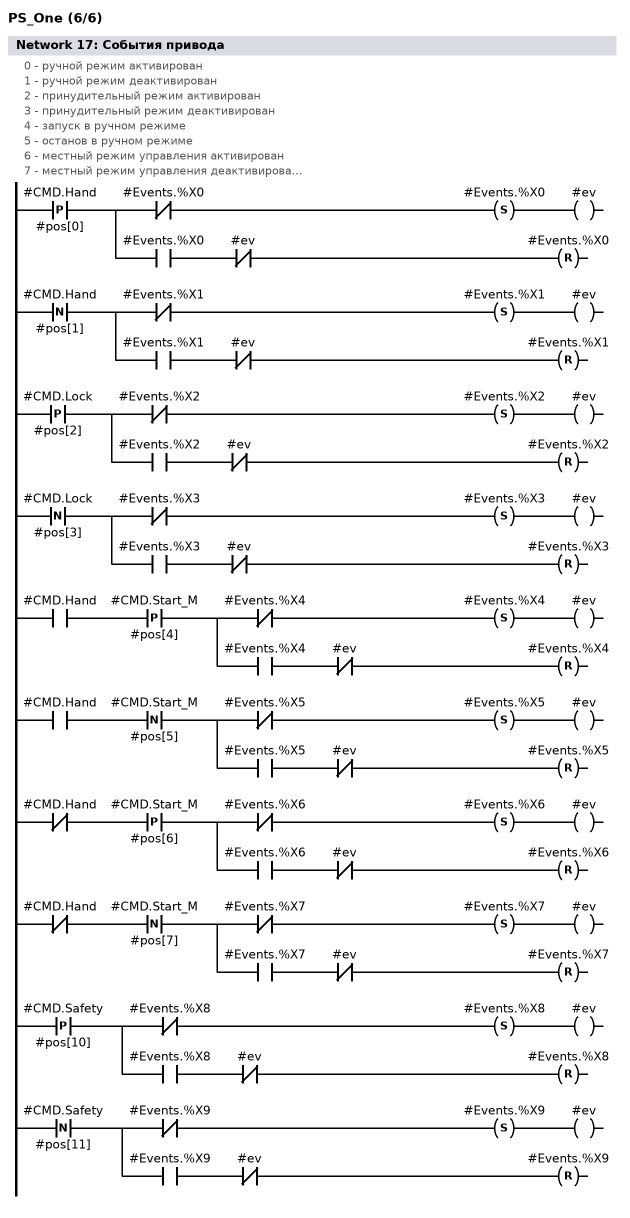
   RUNG wire#powerrail
      P_Contact(operand := #CMD.Hand, bit := #pos[0])
      wire#w1
      I_Contact( #Events.%X0 )
      S_Coil( #Events.%X0 )
      Coil( #ev )
   END_RUNG
   RUNG wire#w1
      Contact( #Events.%X0 )
      I_Contact( #ev )
      R_Coil( #Events.%X0 )
   END_RUNG
   RUNG wire#powerrail
      N_Contact(operand := #CMD.Hand, bit := #pos[1])
      wire#w2
      I_Contact( #Events.%X1 )
      S_Coil( #Events.%X1 )
      Coil( #ev )
   END_RUNG
   RUNG wire#w2
      Contact( #Events.%X1 )
      I_Contact( #ev )
      R_Coil( #Events.%X1 )
   END_RUNG
   RUNG wire#powerrail
      P_Contact(operand := #CMD.Lock, bit := #pos[2])
      wire#w3
      I_Contact( #Events.%X2 )
      S_Coil( #Events.%X2 )
      Coil( #ev )
   END_RUNG
   RUNG wire#w3
      Contact( #Events.%X2 )
      I_Contact( #ev )
      R_Coil( #Events.%X2 )
   END_RUNG
   RUNG wire#powerrail
      N_Contact(operand := #CMD.Lock, bit := #pos[3])
      wire#w4
      I_Contact( #Events.%X3 )
      S_Coil( #Events.%X3 )
      Coil( #ev )
   END_RUNG
   RUNG wire#w4
      Contact( #Events.%X3 )
      I_Contact( #ev )
      R_Coil( #Events.%X3 )
   END_RUNG
   RUNG wire#powerrail
      Contact( #CMD.Hand )
      P_Contact(operand := #CMD.Start_M, bit := #pos[4])
      wire#w5
      I_Contact( #Events.%X4 )
      S_Coil( #Events.%X4 )
      Coil( #ev )
   END_RUNG
   RUNG wire#w5
      Contact( #Events.%X4 )
      I_Contact( #ev )
      R_Coil( #Events.%X4 )
   END_RUNG
   RUNG wire#powerrail
      Contact( #CMD.Hand )
      N_Contact(operand := #CMD.Start_M, bit := #pos[5])
      wire#w6
      I_Contact( #Events.%X5 )
      S_Coil( #Events.%X5 )
      Coil( #ev )
   END_RUNG
   RUNG wire#w6
      Contact( #Events.%X5 )
      I_Contact( #ev )
      R_Coil( #Events.%X5 )
   END_RUNG
   RUNG wire#powerrail
      I_Contact( #CMD.Hand )
      P_Contact(operand := #CMD.Start_M, bit := #pos[6])
      wire#w7
      I_Contact( #Events.%X6 )
      S_Coil( #Events.%X6 )
      Coil( #ev )
   END_RUNG
   RUNG wire#w7
      Contact( #Events.%X6 )
      I_Contact( #ev )
      R_Coil( #Events.%X6 )
   END_RUNG
   RUNG wire#powerrail
      I_Contact( #CMD.Hand )
      N_Contact(operand := #CMD.Start_M, bit := #pos[7])
      wire#w8
      I_Contact( #Events.%X7 )
      S_Coil( #Events.%X7 )
      Coil( #ev )
   END_RUNG
   RUNG wire#w8
      Contact( #Events.%X7 )
      I_Contact( #ev )
      R_Coil( #Events.%X7 )
   END_RUNG
   RUNG wire#powerrail
      P_Contact(operand := #CMD.Safety, bit := #pos[10])
      wire#w9
      I_Contact( #Events.%X8 )
      S_Coil( #Events.%X8 )
      Coil( #ev )
   END_RUNG
   RUNG wire#w9
      Contact( #Events.%X8 )
      I_Contact( #ev )
      R_Coil( #Events.%X8 )
   END_RUNG
   RUNG wire#powerrail
      N_Contact(operand := #CMD.Safety, bit := #pos[11])
      wire#w10
      I_Contact( #Events.%X9 )
      S_Coil( #Events.%X9 )
      Coil( #ev )
   END_RUNG
   RUNG wire#w10
      Contact( #Events.%X9 )
      I_Contact( #ev )
      R_Coil( #Events.%X9 )
   END_RUNG
   // the same network as SCL:
   #_w1 := #CMD.Hand AND NOT #pos[0];   // rising edge of #CMD.Hand
   #pos[0] := #CMD.Hand;
   #_w2 := #_w1 AND NOT #Events.%X0;
   IF #_w2 THEN #Events.%X0 := TRUE; END_IF;
   #ev := #_w2;
   IF #_w1 AND #Events.%X0 AND NOT #ev THEN #Events.%X0 := FALSE; END_IF;
   #_w3 := NOT #CMD.Hand AND #pos[1];   // falling edge of #CMD.Hand
   #pos[1] := #CMD.Hand;
   #_w4 := #_w3 AND NOT #Events.%X1;
   IF #_w4 THEN #Events.%X1 := TRUE; END_IF;
   #ev := #_w4;
   IF #_w3 AND #Events.%X1 AND NOT #ev THEN #Events.%X1 := FALSE; END_IF;
   #_w5 := #CMD.Lock AND NOT #pos[2];   // rising edge of #CMD.Lock
   #pos[2] := #CMD.Lock;
   #_w6 := #_w5 AND NOT #Events.%X2;
   IF #_w6 THEN #Events.%X2 := TRUE; END_IF;
   #ev := #_w6;
   IF #_w5 AND #Events.%X2 AND NOT #ev THEN #Events.%X2 := FALSE; END_IF;
   #_w7 := NOT #CMD.Lock AND #pos[3];   // falling edge of #CMD.Lock
   #pos[3] := #CMD.Lock;
   #_w8 := #_w7 AND NOT #Events.%X3;
   IF #_w8 THEN #Events.%X3 := TRUE; END_IF;
   #ev := #_w8;
   IF #_w7 AND #Events.%X3 AND NOT #ev THEN #Events.%X3 := FALSE; END_IF;
   #_w9 := #CMD.Hand AND #CMD.Start_M AND NOT #pos[4];   // rising edge of #CMD.Start_M
   #pos[4] := #CMD.Start_M;
   #_w10 := #_w9 AND NOT #Events.%X4;
   IF #_w10 THEN #Events.%X4 := TRUE; END_IF;
   #ev := #_w10;
   IF #_w9 AND #Events.%X4 AND NOT #ev THEN #Events.%X4 := FALSE; END_IF;
   #_w11 := #CMD.Hand AND NOT #CMD.Start_M AND #pos[5];   // falling edge of #CMD.Start_M
   #pos[5] := #CMD.Start_M;
   #_w12 := #_w11 AND NOT #Events.%X5;
   IF #_w12 THEN #Events.%X5 := TRUE; END_IF;
   #ev := #_w12;
   IF #_w11 AND #Events.%X5 AND NOT #ev THEN #Events.%X5 := FALSE; END_IF;
   #_w13 := NOT #CMD.Hand AND #CMD.Start_M AND NOT #pos[6];   // rising edge of #CMD.Start_M
   #pos[6] := #CMD.Start_M;
   #_w14 := #_w13 AND NOT #Events.%X6;
   IF #_w14 THEN #Events.%X6 := TRUE; END_IF;
   #ev := #_w14;
   IF #_w13 AND #Events.%X6 AND NOT #ev THEN #Events.%X6 := FALSE; END_IF;
   #_w15 := NOT #CMD.Hand AND NOT #CMD.Start_M AND #pos[7];   // falling edge of #CMD.Start_M
   #pos[7] := #CMD.Start_M;
   #_w16 := #_w15 AND NOT #Events.%X7;
   IF #_w16 THEN #Events.%X7 := TRUE; END_IF;
   #ev := #_w16;
   IF #_w15 AND #Events.%X7 AND NOT #ev THEN #Events.%X7 := FALSE; END_IF;
   #_w17 := #CMD.Safety AND NOT #pos[10];   // rising edge of #CMD.Safety
   #pos[10] := #CMD.Safety;
   #_w18 := #_w17 AND NOT #Events.%X8;
   IF #_w18 THEN #Events.%X8 := TRUE; END_IF;
   #ev := #_w18;
   IF #_w17 AND #Events.%X8 AND NOT #ev THEN #Events.%X8 := FALSE; END_IF;
   #_w19 := NOT #CMD.Safety AND #pos[11];   // falling edge of #CMD.Safety
   #pos[11] := #CMD.Safety;
   #_w20 := #_w19 AND NOT #Events.%X9;
   IF #_w20 THEN #Events.%X9 := TRUE; END_IF;
   #ev := #_w20;
   IF #_w19 AND #Events.%X9 AND NOT #ev THEN #Events.%X9 := FALSE; END_IF;
END_REGION
END_FUNCTION_BLOCK

FUNCTION_BLOCK "Time_D"   // FB94, LAD
{ S7_Optimized_Access := 'FALSE' }
VERSION : 0.1
// stored: AutoNumber false, IsIECCheckEnabled false, SetENOAutomatically false, UDAEnableTagReadback false
   VAR DB_SPECIFIC
      SP_D { S7_SetPoint := 'True'} : DInt := 4;   // Уставка дней - от 0 до 999
      SP_H { S7_SetPoint := 'True'} : DInt;   // Уставка часов - от 0 до 23
      SP_M { S7_SetPoint := 'True'} : DInt;   // Уставка минут - от 0 до 59
      SP_S { S7_SetPoint := 'True'} : DInt;   // Уставка секунд - от 0 до 59
      Now_D : DInt;   // Прошло дней от начала отсчёта
      Now_H : DInt;   // Прошло часов от начала отсчёта
      Now_M : DInt;   // Прошло минут от начала отсчёта
      Now_S : DInt;   // Прошло секунд от начала отсчёта
      Rev_D : DInt;   // Осталось дней до уставки
      Rev_H : DInt;   // Осталось часов до уставки
      Rev_M : DInt;   // Осталось минут до уставки
      Rev_S : DInt;   // Осталось секунд до уставки
      Progress : Real;   // Прогресс выполнения
      Start : Bool;   // Запуск
      "Exit" : Bool;   // Счёт завершён
      Pause : Bool;   // Пауза
      Reset : Bool;   // Сброс таймера
   END_VAR
   VAR_TEMP
      Full_SP_S : DInt;
      Full_Now_S : DInt;
      Full_Delta_S : DInt;
      x1 : DInt;
      x2 : DInt;
   END_VAR
   VAR_TEMP   // added for the SCL form of the ladder/FBD networks
      _w1 : Bool;
      _w2 : Bool;
      _w3 : Bool;
   END_VAR
BEGIN

